LIN {X 0,Y 554.756,Z 744.447,A -85,B 0,C 180,E1 26525.906,E2 26525.906} C_VEL
LIN {X 0,Y 555.497,Z 725.73,A -85,B 0,C 180,E1 26524.354,E2 26524.354} C_VEL
LIN {X 0,Y 556.232,Z 706.632,A -85,B 0,C 180,E1 26523.006,E2 26523.006} C_VEL
LIN {X 0,Y 556.963,Z 686.726,A -85,B 0,C 180,E1 26521.826,E2 26521.826} C_VEL
LIN {X 0,Y 557.64,Z 666.249,A -85,B 0,C 180,E1 26520.833,E2 26520.833} C_VEL
LIN {X 0,Y 558.264,Z 644.541,A -85,B 0,C 180,E1 26519.99,E2 26519.99} C_VEL
LIN {X 0,Y 558.793,Z 623.131,A -85,B 0,C 180,E1 26519.359,E2 26519.359} C_VEL
LIN {X 0,Y 559.115,Z 601.514,A -85,B 0,C 180,E1 26518.923,E2 26518.923} C_VEL
LIN {X 0,Y 560.676,Z 378.924,A -85,B 0,C 180,E1 26515.689,E2 26515.689} C_VEL
LIN {X 0,Y 561.034,Z 312.454,A -85,B 0,C 180,E1 26514.699,E2 26514.699} C_VEL
LIN {X 0,Y 559.13,Z 302.175,A -85,B 0,C 180,E1 26514.381,E2 26514.381} C_VEL
LIN {X 0,Y 560.174,Z 262.496,A -85,B 0,C 180,E1 26511.548,E2 26511.548} C_VEL
LIN {X 0,Y 553.21,Z 246.785,A -85,B 0,C 180,E1 26509.785,E2 26509.785} C_VEL
LIN {X 0,Y 552.322,Z 243.938,A -85,B 0,C 180,E1 26509.493,E2 26509.493} C_VEL
LIN {X 0,Y 552.276,Z 243.94,A -85,B 0,C 180,E1 26506.244,E2 26506.244} C_VEL
LIN {X 0,Y 552.335,Z 243.938,A -85,B 0,C 180,E1 26503.001,E2 26503.001} C_VEL
LIN {X 0,Y 552.275,Z 243.938,A -85,B 0,C 180,E1 26499.858,E2 26499.858} C_VEL
LIN {X 0,Y 552.287,Z 243.939,A -85,B 0,C 180,E1 26496.503,E2 26496.503} C_VEL
LIN {X 0,Y 552.286,Z 243.938,A -85,B 0,C 180,E1 26493.517,E2 26493.517} C_VEL
LIN {X 0,Y 552.27,Z 243.94,A -85,B 0,C 180,E1 26490.22,E2 26490.22} C_VEL
LIN {X 0,Y 552.328,Z 243.939,A -85,B 0,C 180,E1 26487.026,E2 26487.026} C_VEL
LIN {X 0,Y 552.26,Z 243.94,A -85,B 0,C 180,E1 26483.813,E2 26483.813} C_VEL
LIN {X 0,Y 552.351,Z 244.153,A -85,B 0,C 180,E1 26480.713,E2 26480.713} C_VEL
LIN {X 0,Y 553.695,Z 247.553,A -85,B 0,C 180,E1 26480.559,E2 26480.559} C_VEL
LIN {X 0,Y 555.367,Z 250.208,A -85,B 0,C 180,E1 26480.395,E2 26480.395} C_VEL
LIN {X 0,Y 560.988,Z 259.677,A -85,B 0,C 180,E1 26479.842,E2 26479.842} C_VEL
LIN {X 0,Y 559.325,Z 496.337,A -85,B 0,C 180,E1 26476.402,E2 26476.402} C_VEL
LIN {X 0,Y 558.983,Z 531.842,A -85,B 0,C 180,E1 26475.851,E2 26475.851} C_VEL
LIN {X 0,Y 558.554,Z 554.111,A -85,B 0,C 180,E1 26475.298,E2 26475.298} C_VEL
LIN {X 0,Y 557.962,Z 575.135,A -85,B 0,C 180,E1 26474.584,E2 26474.584} C_VEL
LIN {X 0,Y 557.322,Z 596.603,A -85,B 0,C 180,E1 26473.647,E2 26473.647} C_VEL
LIN {X 0,Y 556.604,Z 616.891,A -85,B 0,C 180,E1 26472.555,E2 26472.555} C_VEL
LIN {X 0,Y 555.878,Z 636.118,A -85,B 0,C 180,E1 26471.308,E2 26471.308} C_VEL
LIN {X 0,Y 555.13,Z 655.149,A -85,B 0,C 180,E1 26469.853,E2 26469.853} C_VEL
LIN {X 0,Y 554.42,Z 673.135,A -85,B 0,C 180,E1 26468.244,E2 26468.244} C_VEL
LIN {X 0,Y 553.808,Z 689.545,A -85,B 0,C 180,E1 26466.532,E2 26466.532} C_VEL
LIN {X 0,Y 553.233,Z 705.705,A -85,B 0,C 180,E1 26464.562,E2 26464.562} C_VEL
LIN {X 0,Y 552.797,Z 719.52,A -85,B 0,C 180,E1 26462.593,E2 26462.593} C_VEL
LIN {X 0,Y 552.451,Z 732.51,A -85,B 0,C 180,E1 26460.416,E2 26460.416} C_VEL
LIN {X 0,Y 552.222,Z 742.951,A -85,B 0,C 180,E1 26458.341,E2 26458.341} C_VEL
LIN {X 0,Y 552.065,Z 752.001,A -85,B 0,C 180,E1 26456.159,E2 26456.159} C_VEL
LIN {X 0,Y 551.98,Z 759.324,A -85,B 0,C 180,E1 26453.968,E2 26453.968} C_VEL
LIN {X 0,Y 551.934,Z 765.028,A -85,B 0,C 180,E1 26451.774,E2 26451.774} C_VEL
LIN {X 0,Y 551.912,Z 769.059,A -85,B 0,C 180,E1 26449.564,E2 26449.564} C_VEL
LIN {X 0,Y 551.914,Z 771.636,A -85,B 0,C 180,E1 26447.233,E2 26447.233} C_VEL
LIN {X 0,Y 551.917,Z 772.498,A -85,B 0,C 180,E1 26444.988,E2 26444.988} C_VEL
LIN {X 0,Y 551.911,Z 771.649,A -85,B 0,C 180,E1 26442.695,E2 26442.695} C_VEL
LIN {X 0,Y 551.919,Z 769.139,A -85,B 0,C 180,E1 26440.397,E2 26440.397} C_VEL
LIN {X 0,Y 551.937,Z 765.18,A -85,B 0,C 180,E1 26438.202,E2 26438.202} C_VEL
LIN {X 0,Y 551.98,Z 759.253,A -85,B 0,C 180,E1 26435.917,E2 26435.917} C_VEL
LIN {X 0,Y 552.069,Z 751.656,A -85,B 0,C 180,E1 26433.661,E2 26433.661} C_VEL
LIN {X 0,Y 552.082,Z 750.625,A -85,B 0,C 180,E1 26433.393,E2 26433.393} C_VEL
LIN {X 0,Y 551.135,Z 747.773,A -85,B 0,C 180,E1 26432.65,E2 26432.65} C_VEL
LIN {X 0,Y 545.095,Z 739.69,A -85,B 0,C 180,E1 26430.691,E2 26430.691} C_VEL
LIN {X 0,Y 544.423,Z 736.731,A -85,B 0,C 180,E1 26430.065,E2 26430.065} C_VEL
LIN {X 0,Y 544.761,Z 725.174,A -85,B 0,C 180,E1 26427.968,E2 26427.968} C_VEL
LIN {X 0,Y 545.246,Z 711.568,A -85,B 0,C 180,E1 26425.868,E2 26425.868} C_VEL
LIN {X 0,Y 545.854,Z 696.307,A -85,B 0,C 180,E1 26423.859,E2 26423.859} C_VEL
LIN {X 0,Y 546.544,Z 680.23,A -85,B 0,C 180,E1 26422.044,E2 26422.044} C_VEL
LIN {X 0,Y 547.342,Z 662.41,A -85,B 0,C 180,E1 26420.32,E2 26420.32} C_VEL
LIN {X 0,Y 548.174,Z 644.266,A -85,B 0,C 180,E1 26418.821,E2 26418.821} C_VEL
LIN {X 0,Y 549.064,Z 624.441,A -85,B 0,C 180,E1 26417.432,E2 26417.432} C_VEL
LIN {X 0,Y 549.929,Z 603.469,A -85,B 0,C 180,E1 26416.205,E2 26416.205} C_VEL
LIN {X 0,Y 550.725,Z 582.729,A -85,B 0,C 180,E1 26415.22,E2 26415.22} C_VEL
LIN {X 0,Y 551.396,Z 561.172,A -85,B 0,C 180,E1 26414.411,E2 26414.411} C_VEL
LIN {X 0,Y 551.948,Z 539.46,A -85,B 0,C 180,E1 26413.8,E2 26413.8} C_VEL
LIN {X 0,Y 552.347,Z 516.378,A -85,B 0,C 180,E1 26413.364,E2 26413.364} C_VEL
LIN {X 0,Y 554.178,Z 289.23,A -85,B 0,C 180,E1 26410.034,E2 26410.034} C_VEL
LIN {X 0,Y 554.28,Z 262.154,A -85,B 0,C 180,E1 26409.621,E2 26409.621} C_VEL
LIN {X 0,Y 546.205,Z 249.081,A -85,B 0,C 180,E1 26408.81,E2 26408.81} C_VEL
LIN {X 0,Y 544.543,Z 245.843,A -85,B 0,C 180,E1 26408.631,E2 26408.631} C_VEL
LIN {X 0,Y 544.367,Z 244.904,A -85,B 0,C 180,E1 26408.571,E2 26408.571} C_VEL
LIN {X 0,Y 544.403,Z 244.915,A -85,B 0,C 180,E1 26405.19,E2 26405.19} C_VEL
LIN {X 0,Y 544.372,Z 244.923,A -85,B 0,C 180,E1 26401.937,E2 26401.937} C_VEL
LIN {X 0,Y 544.371,Z 244.926,A -85,B 0,C 180,E1 26398.526,E2 26398.526} C_VEL
LIN {X 0,Y 544.404,Z 244.923,A -85,B 0,C 180,E1 26395.221,E2 26395.221} C_VEL
LIN {X 0,Y 544.364,Z 244.922,A -85,B 0,C 180,E1 26391.893,E2 26391.893} C_VEL
LIN {X 0,Y 544.37,Z 244.925,A -85,B 0,C 180,E1 26388.417,E2 26388.417} C_VEL
LIN {X 0,Y 544.405,Z 244.921,A -85,B 0,C 180,E1 26385.118,E2 26385.118} C_VEL
LIN {X 0,Y 544.358,Z 244.922,A -85,B 0,C 180,E1 26381.872,E2 26381.872} C_VEL
LIN {X 0,Y 544.388,Z 244.924,A -85,B 0,C 180,E1 26378.557,E2 26378.557} C_VEL
LIN {X 0,Y 544.384,Z 244.919,A -85,B 0,C 180,E1 26375.27,E2 26375.27} C_VEL
LIN {X 0,Y 544.352,Z 244.922,A -85,B 0,C 180,E1 26371.896,E2 26371.896} C_VEL
LIN {X 0,Y 544.401,Z 244.922,A -85,B 0,C 180,E1 26368.633,E2 26368.633} C_VEL
LIN {X 0,Y 544.361,Z 244.918,A -85,B 0,C 180,E1 26365.366,E2 26365.366} C_VEL
LIN {X 0,Y 544.356,Z 244.922,A -85,B 0,C 180,E1 26361.977,E2 26361.977} C_VEL
LIN {X 0,Y 544.405,Z 244.922,A -85,B 0,C 180,E1 26358.668,E2 26358.668} C_VEL
LIN {X 0,Y 544.347,Z 244.922,A -85,B 0,C 180,E1 26355.427,E2 26355.427} C_VEL
LIN {X 0,Y 544.366,Z 244.925,A -85,B 0,C 180,E1 26352.028,E2 26352.028} C_VEL
LIN {X 0,Y 544.385,Z 244.921,A -85,B 0,C 180,E1 26348.789,E2 26348.789} C_VEL
LIN {X 0,Y 544.343,Z 244.923,A -85,B 0,C 180,E1 26345.475,E2 26345.475} C_VEL
LIN {X 0,Y 544.393,Z 244.924,A -85,B 0,C 180,E1 26342.194,E2 26342.194} C_VEL
LIN {X 0,Y 544.348,Z 244.924,A -85,B 0,C 180,E1 26339.051,E2 26339.051} C_VEL
LIN {X 0,Y 544.344,Z 244.926,A -85,B 0,C 180,E1 26335.556,E2 26335.556} C_VEL
LIN {X 0,Y 544.402,Z 244.922,A -85,B 0,C 180,E1 26332.297,E2 26332.297} C_VEL
LIN {X 0,Y 544.336,Z 244.924,A -85,B 0,C 180,E1 26329.165,E2 26329.165} C_VEL
LIN {X 0,Y 544.381,Z 244.927,A -85,B 0,C 180,E1 26325.887,E2 26325.887} C_VEL
LIN {X 0,Y 544.35,Z 244.924,A -85,B 0,C 180,E1 26322.667,E2 26322.667} C_VEL
LIN {X 0,Y 544.337,Z 244.924,A -85,B 0,C 180,E1 26319.321,E2 26319.321} C_VEL
LIN {X 0,Y 544.394,Z 244.926,A -85,B 0,C 180,E1 26316.123,E2 26316.123} C_VEL
LIN {X 0,Y 544.329,Z 244.926,A -85,B 0,C 180,E1 26312.921,E2 26312.921} C_VEL
LIN {X 0,Y 544.367,Z 244.926,A -85,B 0,C 180,E1 26309.607,E2 26309.607} C_VEL
LIN {X 0,Y 544.339,Z 244.925,A -85,B 0,C 180,E1 26306.507,E2 26306.507} C_VEL
LIN {X 0,Y 544.333,Z 244.926,A -85,B 0,C 180,E1 26303.145,E2 26303.145} C_VEL
LIN {X 0,Y 544.38,Z 244.925,A -85,B 0,C 180,E1 26299.974,E2 26299.974} C_VEL
LIN {X 0,Y 544.322,Z 244.926,A -85,B 0,C 180,E1 26296.76,E2 26296.76} C_VEL
LIN {X 0,Y 544.386,Z 244.927,A -85,B 0,C 180,E1 26293.595,E2 26293.595} C_VEL
LIN {X 0,Y 544.326,Z 244.925,A -85,B 0,C 180,E1 26290.369,E2 26290.369} C_VEL
LIN {X 0,Y 544.328,Z 244.926,A -85,B 0,C 180,E1 26286.962,E2 26286.962} C_VEL
LIN {X 0,Y 544.368,Z 244.927,A -85,B 0,C 180,E1 26283.79,E2 26283.79} C_VEL
LIN {X 0,Y 544.319,Z 244.925,A -85,B 0,C 180,E1 26280.63,E2 26280.63} C_VEL
LIN {X 0,Y 544.389,Z 244.926,A -85,B 0,C 180,E1 26277.472,E2 26277.472} C_VEL
LIN {X 0,Y 544.325,Z 244.925,A -85,B 0,C 180,E1 26274.2,E2 26274.2} C_VEL
LIN {X 0,Y 544.339,Z 244.926,A -85,B 0,C 180,E1 26270.803,E2 26270.803} C_VEL
LIN {X 0,Y 544.358,Z 244.926,A -85,B 0,C 180,E1 26267.697,E2 26267.697} C_VEL
LIN {X 0,Y 544.327,Z 244.926,A -85,B 0,C 180,E1 26264.443,E2 26264.443} C_VEL
LIN {X 0,Y 544.396,Z 244.924,A -85,B 0,C 180,E1 26261.251,E2 26261.251} C_VEL
LIN {X 0,Y 544.331,Z 244.925,A -85,B 0,C 180,E1 26257.992,E2 26257.992} C_VEL
LIN {X 0,Y 544.351,Z 244.924,A -85,B 0,C 180,E1 26254.645,E2 26254.645} C_VEL
LIN {X 0,Y 544.352,Z 244.926,A -85,B 0,C 180,E1 26251.592,E2 26251.592} C_VEL
LIN {X 0,Y 544.337,Z 244.926,A -85,B 0,C 180,E1 26248.258,E2 26248.258} C_VEL
LIN {X 0,Y 544.405,Z 244.925,A -85,B 0,C 180,E1 26244.995,E2 26244.995} C_VEL
LIN {X 0,Y 544.339,Z 244.926,A -85,B 0,C 180,E1 26241.755,E2 26241.755} C_VEL
LIN {X 0,Y 544.354,Z 244.927,A -85,B 0,C 180,E1 26238.378,E2 26238.378} C_VEL
LIN {X 0,Y 544.381,Z 244.929,A -85,B 0,C 180,E1 26235.147,E2 26235.147} C_VEL
LIN {X 0,Y 544.34,Z 244.929,A -85,B 0,C 180,E1 26231.816,E2 26231.816} C_VEL
LIN {X 0,Y 544.395,Z 245.017,A -85,B 0,C 180,E1 26231.093,E2 26231.093} C_VEL
LIN {X 0,Y 548.823,Z 255.605,A -85,B 0,C 180,E1 26229.915,E2 26229.915} C_VEL
LIN {X 0,Y 553.412,Z 266.114,A -85,B 0,C 180,E1 26228.734,E2 26228.734} C_VEL
LIN {X 0,Y 552.412,Z 303.163,A -85,B 0,C 180,E1 26226.083,E2 26226.083} C_VEL
LIN {X 0,Y 554.642,Z 315.9,A -85,B 0,C 180,E1 26225.716,E2 26225.716} C_VEL
LIN {X 0,Y 552.802,Z 536.145,A -85,B 0,C 180,E1 26222.466,E2 26222.466} C_VEL
LIN {X 0,Y 552.177,Z 609.441,A -85,B 0,C 180,E1 26221.37,E2 26221.37} C_VEL
LIN {X 0,Y 551.642,Z 631.09,A -85,B 0,C 180,E1 26220.851,E2 26220.851} C_VEL
LIN {X 0,Y 551.021,Z 653.26,A -85,B 0,C 180,E1 26220.113,E2 26220.113} C_VEL
LIN {X 0,Y 550.331,Z 673.419,A -85,B 0,C 180,E1 26219.255,E2 26219.255} C_VEL
LIN {X 0,Y 549.499,Z 693.774,A -85,B 0,C 180,E1 26218.174,E2 26218.174} C_VEL
LIN {X 0,Y 548.621,Z 714.159,A -85,B 0,C 180,E1 26216.869,E2 26216.869} C_VEL
LIN {X 0,Y 547.765,Z 732.883,A -85,B 0,C 180,E1 26215.45,E2 26215.45} C_VEL
LIN {X 0,Y 546.978,Z 750.522,A -85,B 0,C 180,E1 26213.883,E2 26213.883} C_VEL
LIN {X 0,Y 546.248,Z 766.698,A -85,B 0,C 180,E1 26212.207,E2 26212.207} C_VEL
LIN {X 0,Y 545.572,Z 782.882,A -85,B 0,C 180,E1 26210.264,E2 26210.264} C_VEL
LIN {X 0,Y 545.042,Z 797.053,A -85,B 0,C 180,E1 26208.281,E2 26208.281} C_VEL
LIN {X 0,Y 544.625,Z 809.74,A -85,B 0,C 180,E1 26206.202,E2 26206.202} C_VEL
LIN {X 0,Y 544.322,Z 820.534,A -85,B 0,C 180,E1 26204.099,E2 26204.099} C_VEL
LIN {X 0,Y 544.119,Z 830.074,A -85,B 0,C 180,E1 26201.876,E2 26201.876} C_VEL
LIN {X 0,Y 544.002,Z 837.94,A -85,B 0,C 180,E1 26199.627,E2 26199.627} C_VEL
LIN {X 0,Y 543.941,Z 843.91,A -85,B 0,C 180,E1 26197.392,E2 26197.392} C_VEL
LIN {X 0,Y 543.921,Z 848.466,A -85,B 0,C 180,E1 26195.061,E2 26195.061} C_VEL
LIN {X 0,Y 543.91,Z 851.236,A -85,B 0,C 180,E1 26192.844,E2 26192.844} C_VEL
LIN {X 0,Y 543.899,Z 852.373,A -85,B 0,C 180,E1 26190.631,E2 26190.631} C_VEL
LIN {X 0,Y 543.899,Z 852.015,A -85,B 0,C 180,E1 26188.313,E2 26188.313} C_VEL
LIN {X 0,Y 543.906,Z 850.219,A -85,B 0,C 180,E1 26186.204,E2 26186.204} C_VEL
LIN {X 0,Y 543.925,Z 846.601,A -85,B 0,C 180,E1 26183.879,E2 26183.879} C_VEL
LIN {X 0,Y 543.965,Z 841.58,A -85,B 0,C 180,E1 26181.65,E2 26181.65} C_VEL
LIN {X 0,Y 544.041,Z 835.043,A -85,B 0,C 180,E1 26179.496,E2 26179.496} C_VEL
LIN {X 0,Y 544.194,Z 826.137,A -85,B 0,C 180,E1 26177.154,E2 26177.154} C_VEL
LIN {X 0,Y 544.438,Z 816.112,A -85,B 0,C 180,E1 26174.992,E2 26174.992} C_VEL
LIN {X 0,Y 544.779,Z 804.625,A -85,B 0,C 180,E1 26172.922,E2 26172.922} C_VEL
LIN {X 0,Y 545.233,Z 791.785,A -85,B 0,C 180,E1 26170.948,E2 26170.948} C_VEL
LIN {X 0,Y 545.792,Z 777.648,A -85,B 0,C 180,E1 26169.069,E2 26169.069} C_VEL
LIN {X 0,Y 546.482,Z 761.672,A -85,B 0,C 180,E1 26167.24,E2 26167.24} C_VEL
LIN {X 0,Y 547.232,Z 744.445,A -85,B 0,C 180,E1 26165.553,E2 26165.553} C_VEL
LIN {X 0,Y 548.104,Z 725.658,A -85,B 0,C 180,E1 26163.977,E2 26163.977} C_VEL
LIN {X 0,Y 548.959,Z 706.635,A -85,B 0,C 180,E1 26162.619,E2 26162.619} C_VEL
LIN {X 0,Y 549.764,Z 687.244,A -85,B 0,C 180,E1 26161.454,E2 26161.454} C_VEL
LIN {X 0,Y 550.55,Z 666.868,A -85,B 0,C 180,E1 26160.449,E2 26160.449} C_VEL
LIN {X 0,Y 551.261,Z 645.621,A -85,B 0,C 180,E1 26159.606,E2 26159.606} C_VEL
LIN {X 0,Y 551.832,Z 624.803,A -85,B 0,C 180,E1 26158.978,E2 26158.978} C_VEL
LIN {X 0,Y 552.243,Z 602.978,A -85,B 0,C 180,E1 26158.519,E2 26158.519} C_VEL
LIN {X 0,Y 554.054,Z 380.884,A -85,B 0,C 180,E1 26155.251,E2 26155.251} C_VEL
LIN {X 0,Y 554.471,Z 313.922,A -85,B 0,C 180,E1 26154.24,E2 26154.24} C_VEL
LIN {X 0,Y 552.308,Z 302.396,A -85,B 0,C 180,E1 26153.888,E2 26153.888} C_VEL
LIN {X 0,Y 553.412,Z 266.114,A -85,B 0,C 180,E1 26151.266,E2 26151.266} C_VEL
LIN {X 0,Y 548.725,Z 255.516,A -85,B 0,C 180,E1 26150.097,E2 26150.097} C_VEL
LIN {X 0,Y 544.489,Z 245.476,A -85,B 0,C 180,E1 26149.092,E2 26149.092} C_VEL
LIN {X 0,Y 544.394,Z 244.927,A -85,B 0,C 180,E1 26149.014,E2 26149.014} C_VEL
LIN {X 0,Y 544.35,Z 244.928,A -85,B 0,C 180,E1 26145.754,E2 26145.754} C_VEL
LIN {X 0,Y 544.34,Z 244.929,A -85,B 0,C 180,E1 26142.386,E2 26142.386} C_VEL
LIN {X 0,Y 544.398,Z 244.926,A -85,B 0,C 180,E1 26139.184,E2 26139.184} C_VEL
LIN {X 0,Y 544.332,Z 244.928,A -85,B 0,C 180,E1 26135.898,E2 26135.898} C_VEL
LIN {X 0,Y 544.352,Z 244.929,A -85,B 0,C 180,E1 26132.532,E2 26132.532} C_VEL
LIN {X 0,Y 544.345,Z 244.929,A -85,B 0,C 180,E1 26129.465,E2 26129.465} C_VEL
LIN {X 0,Y 544.328,Z 244.93,A -85,B 0,C 180,E1 26126.159,E2 26126.159} C_VEL
LIN {X 0,Y 544.395,Z 244.927,A -85,B 0,C 180,E1 26122.916,E2 26122.916} C_VEL
LIN {X 0,Y 544.377,Z 245.171,A -85,B 0,C 180,E1 26121.303,E2 26121.303} C_VEL
LIN {X 0,Y 545.785,Z 248.582,A -85,B 0,C 180,E1 26121.14,E2 26121.14} C_VEL
LIN {X 0,Y 547.429,Z 251.037,A -85,B 0,C 180,E1 26120.975,E2 26120.975} C_VEL
LIN {X 0,Y 554.403,Z 262.797,A -85,B 0,C 180,E1 26120.27,E2 26120.27} C_VEL
LIN {X 0,Y 552.475,Z 500.076,A -85,B 0,C 180,E1 26116.781,E2 26116.781} C_VEL
LIN {X 0,Y 552.096,Z 532.411,A -85,B 0,C 180,E1 26116.266,E2 26116.266} C_VEL
LIN {X 0,Y 551.595,Z 554.888,A -85,B 0,C 180,E1 26115.698,E2 26115.698} C_VEL
LIN {X 0,Y 550.916,Z 576.092,A -85,B 0,C 180,E1 26114.963,E2 26114.963} C_VEL
LIN {X 0,Y 550.195,Z 596.838,A -85,B 0,C 180,E1 26114.042,E2 26114.042} C_VEL
LIN {X 0,Y 549.368,Z 617.108,A -85,B 0,C 180,E1 26112.937,E2 26112.937} C_VEL
LIN {X 0,Y 548.502,Z 637.055,A -85,B 0,C 180,E1 26111.622,E2 26111.622} C_VEL
LIN {X 0,Y 547.634,Z 655.942,A -85,B 0,C 180,E1 26110.149,E2 26110.149} C_VEL
LIN {X 0,Y 546.795,Z 674.342,A -85,B 0,C 180,E1 26108.466,E2 26108.466} C_VEL
LIN {X 0,Y 546.093,Z 690.578,A -85,B 0,C 180,E1 26106.731,E2 26106.731} C_VEL
LIN {X 0,Y 545.437,Z 706.62,A -85,B 0,C 180,E1 26104.733,E2 26104.733} C_VEL
LIN {X 0,Y 544.931,Z 720.295,A -85,B 0,C 180,E1 26102.736,E2 26102.736} C_VEL
LIN {X 0,Y 544.544,Z 732.587,A -85,B 0,C 180,E1 26100.633,E2 26100.633} C_VEL
LIN {X 0,Y 544.266,Z 743.479,A -85,B 0,C 180,E1 26098.422,E2 26098.422} C_VEL
LIN {X 0,Y 544.088,Z 752.449,A -85,B 0,C 180,E1 26096.208,E2 26096.208} C_VEL
LIN {X 0,Y 543.986,Z 759.844,A -85,B 0,C 180,E1 26093.92,E2 26093.92} C_VEL
LIN {X 0,Y 543.939,Z 765.497,A -85,B 0,C 180,E1 26091.652,E2 26091.652} C_VEL
LIN {X 0,Y 543.917,Z 769.397,A -85,B 0,C 180,E1 26089.409,E2 26089.409} C_VEL
LIN {X 0,Y 543.908,Z 771.782,A -85,B 0,C 180,E1 26087.042,E2 26087.042} C_VEL
LIN {X 0,Y 543.905,Z 772.474,A -85,B 0,C 180,E1 26084.761,E2 26084.761} C_VEL
LIN {X 0,Y 543.907,Z 771.513,A -85,B 0,C 180,E1 26082.455,E2 26082.455} C_VEL
LIN {X 0,Y 543.918,Z 768.828,A -85,B 0,C 180,E1 26080.12,E2 26080.12} C_VEL
LIN {X 0,Y 543.933,Z 764.644,A -85,B 0,C 180,E1 26077.865,E2 26077.865} C_VEL
LIN {X 0,Y 543.992,Z 758.658,A -85,B 0,C 180,E1 26075.574,E2 26075.574} C_VEL
LIN {X 0,Y 544.106,Z 751.164,A -85,B 0,C 180,E1 26073.363,E2 26073.363} C_VEL
LIN {X 0,Y 544.301,Z 741.783,A -85,B 0,C 180,E1 26071.113,E2 26071.113} C_VEL
LIN {X 0,Y 544.423,Z 736.731,A -85,B 0,C 180,E1 26070.065,E2 26070.065} C_VEL
LIN {X 0,Y 543.541,Z 733.191,A -85,B 0,C 180,E1 26069.343,E2 26069.343} C_VEL
LIN {X 0,Y 537.721,Z 723.441,A -85,B 0,C 180,E1 26067.437,E2 26067.437} C_VEL
LIN {X 0,Y 537.11,Z 719.871,A -85,B 0,C 180,E1 26066.839,E2 26066.839} C_VEL
LIN {X 0,Y 537.708,Z 706.045,A -85,B 0,C 180,E1 26064.802,E2 26064.802} C_VEL
LIN {X 0,Y 538.457,Z 690.185,A -85,B 0,C 180,E1 26062.808,E2 26062.808} C_VEL
LIN {X 0,Y 539.317,Z 673.099,A -85,B 0,C 180,E1 26060.969,E2 26060.969} C_VEL
LIN {X 0,Y 540.255,Z 654.693,A -85,B 0,C 180,E1 26059.282,E2 26059.282} C_VEL
LIN {X 0,Y 541.252,Z 635.649,A -85,B 0,C 180,E1 26057.798,E2 26057.798} C_VEL
LIN {X 0,Y 542.197,Z 616.697,A -85,B 0,C 180,E1 26056.544,E2 26056.544} C_VEL
LIN {X 0,Y 543.16,Z 595.704,A -85,B 0,C 180,E1 26055.394,E2 26055.394} C_VEL
LIN {X 0,Y 544.026,Z 574.141,A -85,B 0,C 180,E1 26054.447,E2 26054.447} C_VEL
LIN {X 0,Y 544.72,Z 552.664,A -85,B 0,C 180,E1 26053.712,E2 26053.712} C_VEL
LIN {X 0,Y 545.299,Z 530.695,A -85,B 0,C 180,E1 26053.171,E2 26053.171} C_VEL
LIN {X 0,Y 545.781,Z 488.239,A -85,B 0,C 180,E1 26052.511,E2 26052.511} C_VEL
LIN {X 0,Y 547.822,Z 265.586,A -85,B 0,C 180,E1 26049.195,E2 26049.195} C_VEL
LIN {X 0,Y 538.295,Z 250.11,A -85,B 0,C 180,E1 26048.21,E2 26048.21} C_VEL
LIN {X 0,Y 536.619,Z 246.873,A -85,B 0,C 180,E1 26048.023,E2 26048.023} C_VEL
LIN {X 0,Y 536.434,Z 245.877,A -85,B 0,C 180,E1 26047.965,E2 26047.965} C_VEL
LIN {X 0,Y 536.429,Z 245.916,A -85,B 0,C 180,E1 26044.516,E2 26044.516} C_VEL
LIN {X 0,Y 536.466,Z 245.914,A -85,B 0,C 180,E1 26041.193,E2 26041.193} C_VEL
LIN {X 0,Y 536.432,Z 245.912,A -85,B 0,C 180,E1 26037.895,E2 26037.895} C_VEL
LIN {X 0,Y 536.43,Z 245.915,A -85,B 0,C 180,E1 26034.444,E2 26034.444} C_VEL
LIN {X 0,Y 536.467,Z 245.912,A -85,B 0,C 180,E1 26031.083,E2 26031.083} C_VEL
LIN {X 0,Y 536.427,Z 245.911,A -85,B 0,C 180,E1 26027.746,E2 26027.746} C_VEL
LIN {X 0,Y 536.423,Z 245.911,A -85,B 0,C 180,E1 26024.244,E2 26024.244} C_VEL
LIN {X 0,Y 536.465,Z 245.911,A -85,B 0,C 180,E1 26020.96,E2 26020.96} C_VEL
LIN {X 0,Y 536.417,Z 245.911,A -85,B 0,C 180,E1 26017.714,E2 26017.714} C_VEL
LIN {X 0,Y 536.43,Z 245.913,A -85,B 0,C 180,E1 26014.277,E2 26014.277} C_VEL
LIN {X 0,Y 536.463,Z 245.908,A -85,B 0,C 180,E1 26010.962,E2 26010.962} C_VEL
LIN {X 0,Y 536.414,Z 245.911,A -85,B 0,C 180,E1 26007.651,E2 26007.651} C_VEL
LIN {X 0,Y 536.433,Z 245.913,A -85,B 0,C 180,E1 26004.224,E2 26004.224} C_VEL
LIN {X 0,Y 536.446,Z 245.907,A -85,B 0,C 180,E1 26000.994,E2 26000.994} C_VEL
LIN {X 0,Y 536.409,Z 245.911,A -85,B 0,C 180,E1 25997.623,E2 25997.623} C_VEL
LIN {X 0,Y 536.453,Z 245.912,A -85,B 0,C 180,E1 25994.322,E2 25994.322} C_VEL
LIN {X 0,Y 536.423,Z 245.911,A -85,B 0,C 180,E1 25991.077,E2 25991.077} C_VEL
LIN {X 0,Y 536.407,Z 245.913,A -85,B 0,C 180,E1 25987.652,E2 25987.652} C_VEL
LIN {X 0,Y 536.464,Z 245.913,A -85,B 0,C 180,E1 25984.382,E2 25984.382} C_VEL
LIN {X 0,Y 536.408,Z 245.911,A -85,B 0,C 180,E1 25981.135,E2 25981.135} C_VEL
LIN {X 0,Y 536.409,Z 245.912,A -85,B 0,C 180,E1 25977.66,E2 25977.66} C_VEL
LIN {X 0,Y 536.461,Z 245.914,A -85,B 0,C 180,E1 25974.348,E2 25974.348} C_VEL
LIN {X 0,Y 536.4,Z 245.915,A -85,B 0,C 180,E1 25971.086,E2 25971.086} C_VEL
LIN {X 0,Y 536.419,Z 245.916,A -85,B 0,C 180,E1 25967.712,E2 25967.712} C_VEL
LIN {X 0,Y 536.432,Z 245.913,A -85,B 0,C 180,E1 25964.49,E2 25964.49} C_VEL
LIN {X 0,Y 536.395,Z 245.915,A -85,B 0,C 180,E1 25961.145,E2 25961.145} C_VEL
LIN {X 0,Y 536.458,Z 245.915,A -85,B 0,C 180,E1 25957.953,E2 25957.953} C_VEL
LIN {X 0,Y 536.399,Z 245.911,A -85,B 0,C 180,E1 25954.714,E2 25954.714} C_VEL
LIN {X 0,Y 536.395,Z 245.914,A -85,B 0,C 180,E1 25951.209,E2 25951.209} C_VEL
LIN {X 0,Y 536.454,Z 245.914,A -85,B 0,C 180,E1 25948.011,E2 25948.011} C_VEL
LIN {X 0,Y 536.388,Z 245.913,A -85,B 0,C 180,E1 25944.795,E2 25944.795} C_VEL
LIN {X 0,Y 536.43,Z 245.915,A -85,B 0,C 180,E1 25941.54,E2 25941.54} C_VEL
LIN {X 0,Y 536.398,Z 245.915,A -85,B 0,C 180,E1 25938.36,E2 25938.36} C_VEL
LIN {X 0,Y 536.391,Z 245.915,A -85,B 0,C 180,E1 25935.015,E2 25935.015} C_VEL
LIN {X 0,Y 536.44,Z 245.916,A -85,B 0,C 180,E1 25931.829,E2 25931.829} C_VEL
LIN {X 0,Y 536.38,Z 245.916,A -85,B 0,C 180,E1 25928.575,E2 25928.575} C_VEL
LIN {X 0,Y 536.427,Z 245.916,A -85,B 0,C 180,E1 25925.346,E2 25925.346} C_VEL
LIN {X 0,Y 536.393,Z 245.917,A -85,B 0,C 180,E1 25922.135,E2 25922.135} C_VEL
LIN {X 0,Y 536.385,Z 245.916,A -85,B 0,C 180,E1 25918.717,E2 25918.717} C_VEL
LIN {X 0,Y 536.448,Z 245.917,A -85,B 0,C 180,E1 25915.509,E2 25915.509} C_VEL
LIN {X 0,Y 536.385,Z 245.916,A -85,B 0,C 180,E1 25912.286,E2 25912.286} C_VEL
LIN {X 0,Y 536.414,Z 245.914,A -85,B 0,C 180,E1 25908.93,E2 25908.93} C_VEL
LIN {X 0,Y 536.413,Z 245.915,A -85,B 0,C 180,E1 25905.751,E2 25905.751} C_VEL
LIN {X 0,Y 536.391,Z 245.915,A -85,B 0,C 180,E1 25902.423,E2 25902.423} C_VEL
LIN {X 0,Y 536.458,Z 245.912,A -85,B 0,C 180,E1 25899.145,E2 25899.145} C_VEL
LIN {X 0,Y 536.397,Z 245.914,A -85,B 0,C 180,E1 25895.906,E2 25895.906} C_VEL
LIN {X 0,Y 536.403,Z 245.913,A -85,B 0,C 180,E1 25892.465,E2 25892.465} C_VEL
LIN {X 0,Y 536.452,Z 245.916,A -85,B 0,C 180,E1 25889.227,E2 25889.227} C_VEL
LIN {X 0,Y 536.396,Z 245.916,A -85,B 0,C 180,E1 25885.998,E2 25885.998} C_VEL
LIN {X 0,Y 536.441,Z 245.913,A -85,B 0,C 180,E1 25882.716,E2 25882.716} C_VEL
LIN {X 0,Y 536.41,Z 245.917,A -85,B 0,C 180,E1 25879.558,E2 25879.558} C_VEL
LIN {X 0,Y 536.404,Z 245.918,A -85,B 0,C 180,E1 25876.099,E2 25876.099} C_VEL
LIN {X 0,Y 536.463,Z 245.915,A -85,B 0,C 180,E1 25872.864,E2 25872.864} C_VEL
LIN {X 0,Y 536.404,Z 245.933,A -85,B 0,C 180,E1 25871.715,E2 25871.715} C_VEL
LIN {X 0,Y 537.789,Z 249.492,A -85,B 0,C 180,E1 25871.312,E2 25871.312} C_VEL
LIN {X 0,Y 546.668,Z 269.771,A -85,B 0,C 180,E1 25869.02,E2 25869.02} C_VEL
LIN {X 0,Y 545.621,Z 303.108,A -85,B 0,C 180,E1 25866.605,E2 25866.605} C_VEL
LIN {X 0,Y 548.131,Z 317.548,A -85,B 0,C 180,E1 25866.181,E2 25866.181} C_VEL
LIN {X 0,Y 546.036,Z 538.054,A -85,B 0,C 180,E1 25862.889,E2 25862.889} C_VEL
LIN {X 0,Y 545.342,Z 609.441,A -85,B 0,C 180,E1 25861.809,E2 25861.809} C_VEL
LIN {X 0,Y 544.741,Z 631.09,A -85,B 0,C 180,E1 25861.285,E2 25861.285} C_VEL
LIN {X 0,Y 544.046,Z 653.257,A -85,B 0,C 180,E1 25860.539,E2 25860.539} C_VEL
LIN {X 0,Y 543.253,Z 673.418,A -85,B 0,C 180,E1 25859.674,E2 25859.674} C_VEL
LIN {X 0,Y 542.321,Z 693.777,A -85,B 0,C 180,E1 25858.581,E2 25858.581} C_VEL
LIN {X 0,Y 541.316,Z 714.156,A -85,B 0,C 180,E1 25857.262,E2 25857.262} C_VEL
LIN {X 0,Y 540.362,Z 732.791,A -85,B 0,C 180,E1 25855.832,E2 25855.832} C_VEL
LIN {X 0,Y 539.448,Z 750.621,A -85,B 0,C 180,E1 25854.228,E2 25854.228} C_VEL
LIN {X 0,Y 538.586,Z 767.204,A -85,B 0,C 180,E1 25852.483,E2 25852.483} C_VEL
LIN {X 0,Y 537.832,Z 782.883,A -85,B 0,C 180,E1 25850.569,E2 25850.569} C_VEL
LIN {X 0,Y 537.225,Z 797.054,A -85,B 0,C 180,E1 25848.556,E2 25848.556} C_VEL
LIN {X 0,Y 536.747,Z 809.739,A -85,B 0,C 180,E1 25846.447,E2 25846.447} C_VEL
LIN {X 0,Y 536.402,Z 820.339,A -85,B 0,C 180,E1 25844.353,E2 25844.353} C_VEL
LIN {X 0,Y 536.157,Z 830.074,A -85,B 0,C 180,E1 25842.055,E2 25842.055} C_VEL
LIN {X 0,Y 536.018,Z 837.94,A -85,B 0,C 180,E1 25839.772,E2 25839.772} C_VEL
LIN {X 0,Y 535.945,Z 843.91,A -85,B 0,C 180,E1 25837.503,E2 25837.503} C_VEL
LIN {X 0,Y 535.923,Z 848.465,A -85,B 0,C 180,E1 25835.137,E2 25835.137} C_VEL
LIN {X 0,Y 535.911,Z 851.236,A -85,B 0,C 180,E1 25832.886,E2 25832.886} C_VEL
LIN {X 0,Y 535.899,Z 852.373,A -85,B 0,C 180,E1 25830.64,E2 25830.64} C_VEL
LIN {X 0,Y 535.9,Z 852.015,A -85,B 0,C 180,E1 25828.288,E2 25828.288} C_VEL
LIN {X 0,Y 535.908,Z 850.219,A -85,B 0,C 180,E1 25826.148,E2 25826.148} C_VEL
LIN {X 0,Y 535.926,Z 846.601,A -85,B 0,C 180,E1 25823.787,E2 25823.787} C_VEL
LIN {X 0,Y 535.968,Z 841.58,A -85,B 0,C 180,E1 25821.524,E2 25821.524} C_VEL
LIN {X 0,Y 536.059,Z 835.109,A -85,B 0,C 180,E1 25819.358,E2 25819.358} C_VEL
LIN {X 0,Y 536.233,Z 826.595,A -85,B 0,C 180,E1 25817.07,E2 25817.07} C_VEL
LIN {X 0,Y 536.512,Z 816.682,A -85,B 0,C 180,E1 25814.875,E2 25814.875} C_VEL
LIN {X 0,Y 536.895,Z 805.267,A -85,B 0,C 180,E1 25812.775,E2 25812.775} C_VEL
LIN {X 0,Y 537.446,Z 791.784,A -85,B 0,C 180,E1 25810.661,E2 25810.661} C_VEL
LIN {X 0,Y 538.093,Z 777.647,A -85,B 0,C 180,E1 25808.755,E2 25808.755} C_VEL
LIN {X 0,Y 538.888,Z 761.611,A -85,B 0,C 180,E1 25806.894,E2 25806.894} C_VEL
LIN {X 0,Y 539.74,Z 744.456,A -85,B 0,C 180,E1 25805.192,E2 25805.192} C_VEL
LIN {X 0,Y 540.726,Z 725.655,A -85,B 0,C 180,E1 25803.595,E2 25803.595} C_VEL
LIN {X 0,Y 541.712,Z 706.638,A -85,B 0,C 180,E1 25802.221,E2 25802.221} C_VEL
LIN {X 0,Y 542.582,Z 687.945,A -85,B 0,C 180,E1 25801.083,E2 25801.083} C_VEL
LIN {X 0,Y 543.487,Z 667.479,A -85,B 0,C 180,E1 25800.055,E2 25800.055} C_VEL
LIN {X 0,Y 544.284,Z 646.701,A -85,B 0,C 180,E1 25799.213,E2 25799.213} C_VEL
LIN {X 0,Y 544.919,Z 625.849,A -85,B 0,C 180,E1 25798.571,E2 25798.571} C_VEL
LIN {X 0,Y 545.409,Z 603.622,A -85,B 0,C 180,E1 25798.09,E2 25798.09} C_VEL
LIN {X 0,Y 547.46,Z 383.047,A -85,B 0,C 180,E1 25794.804,E2 25794.804} C_VEL
LIN {X 0,Y 547.95,Z 315.388,A -85,B 0,C 180,E1 25793.771,E2 25793.771} C_VEL
LIN {X 0,Y 545.533,Z 302.117,A -85,B 0,C 180,E1 25793.347,E2 25793.347} C_VEL
LIN {X 0,Y 546.668,Z 269.77,A -85,B 0,C 180,E1 25790.98,E2 25790.98} C_VEL
LIN {X 0,Y 538.015,Z 250.328,A -85,B 0,C 180,E1 25788.984,E2 25788.984} C_VEL
LIN {X 0,Y 536.41,Z 245.92,A -85,B 0,C 180,E1 25788.532,E2 25788.532} C_VEL
LIN {X 0,Y 536.459,Z 245.915,A -85,B 0,C 180,E1 25785.245,E2 25785.245} C_VEL
LIN {X 0,Y 536.398,Z 245.917,A -85,B 0,C 180,E1 25781.948,E2 25781.948} C_VEL
LIN {X 0,Y 536.42,Z 245.918,A -85,B 0,C 180,E1 25778.64,E2 25778.64} C_VEL
LIN {X 0,Y 536.42,Z 245.916,A -85,B 0,C 180,E1 25775.429,E2 25775.429} C_VEL
LIN {X 0,Y 536.39,Z 245.918,A -85,B 0,C 180,E1 25772.091,E2 25772.091} C_VEL
LIN {X 0,Y 536.453,Z 245.916,A -85,B 0,C 180,E1 25768.835,E2 25768.835} C_VEL
LIN {X 0,Y 536.394,Z 245.919,A -85,B 0,C 180,E1 25765.551,E2 25765.551} C_VEL
LIN {X 0,Y 536.388,Z 245.922,A -85,B 0,C 180,E1 25762.113,E2 25762.113} C_VEL
LIN {X 0,Y 536.417,Z 246.171,A -85,B 0,C 180,E1 25761.915,E2 25761.915} C_VEL
LIN {X 0,Y 537.732,Z 249.471,A -85,B 0,C 180,E1 25761.755,E2 25761.755} C_VEL
LIN {X 0,Y 539.482,Z 251.972,A -85,B 0,C 180,E1 25761.576,E2 25761.576} C_VEL
LIN {X 0,Y 547.851,Z 265.911,A -85,B 0,C 180,E1 25760.707,E2 25760.707} C_VEL
LIN {X 0,Y 545.648,Z 504.068,A -85,B 0,C 180,E1 25757.167,E2 25757.167} C_VEL
LIN {X 0,Y 545.234,Z 533.131,A -85,B 0,C 180,E1 25756.689,E2 25756.689} C_VEL
LIN {X 0,Y 544.657,Z 556.001,A -85,B 0,C 180,E1 25756.098,E2 25756.098} C_VEL
LIN {X 0,Y 543.864,Z 577.688,A -85,B 0,C 180,E1 25755.325,E2 25755.325} C_VEL
LIN {X 0,Y 543.047,Z 598.11,A -85,B 0,C 180,E1 25754.394,E2 25754.394} C_VEL
LIN {X 0,Y 542.122,Z 618.21,A -85,B 0,C 180,E1 25753.276,E2 25753.276} C_VEL
LIN {X 0,Y 541.107,Z 638.73,A -85,B 0,C 180,E1 25751.891,E2 25751.891} C_VEL
LIN {X 0,Y 540.125,Z 657.352,A -85,B 0,C 180,E1 25750.399,E2 25750.399} C_VEL
LIN {X 0,Y 539.177,Z 675.532,A -85,B 0,C 180,E1 25748.694,E2 25748.694} C_VEL
LIN {X 0,Y 538.335,Z 692.513,A -85,B 0,C 180,E1 25746.828,E2 25746.828} C_VEL
LIN {X 0,Y 537.641,Z 707.503,A -85,B 0,C 180,E1 25744.909,E2 25744.909} C_VEL
LIN {X 0,Y 537.044,Z 721.721,A -85,B 0,C 180,E1 25742.776,E2 25742.776} C_VEL
LIN {X 0,Y 536.611,Z 733.783,A -85,B 0,C 180,E1 25740.642,E2 25740.642} C_VEL
LIN {X 0,Y 536.287,Z 744.905,A -85,B 0,C 180,E1 25738.292,E2 25738.292} C_VEL
LIN {X 0,Y 536.096,Z 753.636,A -85,B 0,C 180,E1 25736.045,E2 25736.045} C_VEL
LIN {X 0,Y 535.987,Z 760.589,A -85,B 0,C 180,E1 25733.79,E2 25733.79} C_VEL
LIN {X 0,Y 535.936,Z 766.138,A -85,B 0,C 180,E1 25731.418,E2 25731.418} C_VEL
LIN {X 0,Y 535.909,Z 769.851,A -85,B 0,C 180,E1 25729.14,E2 25729.14} C_VEL
LIN {X 0,Y 535.899,Z 771.927,A -85,B 0,C 180,E1 25726.845,E2 25726.845} C_VEL
LIN {X 0,Y 535.906,Z 772.416,A -85,B 0,C 180,E1 25724.417,E2 25724.417} C_VEL
LIN {X 0,Y 535.908,Z 771.247,A -85,B 0,C 180,E1 25722.073,E2 25722.073} C_VEL
LIN {X 0,Y 535.91,Z 768.312,A -85,B 0,C 180,E1 25719.697,E2 25719.697} C_VEL
LIN {X 0,Y 535.939,Z 763.817,A -85,B 0,C 180,E1 25717.401,E2 25717.401} C_VEL
LIN {X 0,Y 536.027,Z 757.576,A -85,B 0,C 180,E1 25715.069,E2 25715.069} C_VEL
LIN {X 0,Y 536.177,Z 749.757,A -85,B 0,C 180,E1 25712.812,E2 25712.812} C_VEL
LIN {X 0,Y 536.424,Z 739.992,A -85,B 0,C 180,E1 25710.525,E2 25710.525} C_VEL
LIN {X 0,Y 536.79,Z 728.673,A -85,B 0,C 180,E1 25708.316,E2 25708.316} C_VEL
LIN {X 0,Y 537.11,Z 719.871,A -85,B 0,C 180,E1 25706.839,E2 25706.839} C_VEL
LIN {X 0,Y 536.295,Z 715.69,A -85,B 0,C 180,E1 25706.149,E2 25706.149} C_VEL
LIN {X 0,Y 530.745,Z 704.443,A -85,B 0,C 180,E1 25704.306,E2 25704.306} C_VEL
LIN {X 0,Y 530.261,Z 700.374,A -85,B 0,C 180,E1 25703.734,E2 25703.734} C_VEL
LIN {X 0,Y 531.123,Z 684.545,A -85,B 0,C 180,E1 25701.827,E2 25701.827} C_VEL
LIN {X 0,Y 532.133,Z 667.051,A -85,B 0,C 180,E1 25700.017,E2 25700.017} C_VEL
LIN {X 0,Y 533.263,Z 648.06,A -85,B 0,C 180,E1 25698.345,E2 25698.345} C_VEL
LIN {X 0,Y 534.358,Z 629.03,A -85,B 0,C 180,E1 25696.927,E2 25696.927} C_VEL
LIN {X 0,Y 535.447,Z 608.76,A -85,B 0,C 180,E1 25695.659,E2 25695.659} C_VEL
LIN {X 0,Y 536.503,Z 587.481,A -85,B 0,C 180,E1 25694.574,E2 25694.574} C_VEL
LIN {X 0,Y 537.422,Z 565.024,A -85,B 0,C 180,E1 25693.666,E2 25693.666} C_VEL
LIN {X 0,Y 538.188,Z 542.413,A -85,B 0,C 180,E1 25692.987,E2 25692.987} C_VEL
LIN {X 0,Y 538.687,Z 520.239,A -85,B 0,C 180,E1 25692.533,E2 25692.533} C_VEL
LIN {X 0,Y 541.031,Z 295.74,A -85,B 0,C 180,E1 25689.161,E2 25689.161} C_VEL
LIN {X 0,Y 541.162,Z 268.343,A -85,B 0,C 180,E1 25688.73,E2 25688.73} C_VEL
LIN {X 0,Y 530.454,Z 251.158,A -85,B 0,C 180,E1 25687.591,E2 25687.591} C_VEL
LIN {X 0,Y 528.732,Z 247.94,A -85,B 0,C 180,E1 25687.393,E2 25687.393} C_VEL
LIN {X 0,Y 528.521,Z 246.855,A -85,B 0,C 180,E1 25687.339,E2 25687.339} C_VEL
LIN {X 0,Y 528.49,Z 246.903,A -85,B 0,C 180,E1 25684.043,E2 25684.043} C_VEL
LIN {X 0,Y 528.497,Z 246.905,A -85,B 0,C 180,E1 25680.593,E2 25680.593} C_VEL
LIN {X 0,Y 528.53,Z 246.901,A -85,B 0,C 180,E1 25677.241,E2 25677.241} C_VEL
LIN {X 0,Y 528.489,Z 246.901,A -85,B 0,C 180,E1 25673.884,E2 25673.884} C_VEL
LIN {X 0,Y 528.488,Z 246.903,A -85,B 0,C 180,E1 25670.373,E2 25670.373} C_VEL
LIN {X 0,Y 528.528,Z 246.901,A -85,B 0,C 180,E1 25667.052,E2 25667.052} C_VEL
LIN {X 0,Y 528.487,Z 246.897,A -85,B 0,C 180,E1 25663.68,E2 25663.68} C_VEL
LIN {X 0,Y 528.486,Z 246.903,A -85,B 0,C 180,E1 25660.245,E2 25660.245} C_VEL
LIN {X 0,Y 528.53,Z 246.9,A -85,B 0,C 180,E1 25656.846,E2 25656.846} C_VEL
LIN {X 0,Y 528.487,Z 246.899,A -85,B 0,C 180,E1 25653.472,E2 25653.472} C_VEL
LIN {X 0,Y 528.479,Z 246.899,A -85,B 0,C 180,E1 25650.001,E2 25650.001} C_VEL
LIN {X 0,Y 528.524,Z 246.902,A -85,B 0,C 180,E1 25646.639,E2 25646.639} C_VEL
LIN {X 0,Y 528.487,Z 246.899,A -85,B 0,C 180,E1 25643.265,E2 25643.265} C_VEL
LIN {X 0,Y 528.475,Z 246.901,A -85,B 0,C 180,E1 25639.867,E2 25639.867} C_VEL
LIN {X 0,Y 528.528,Z 246.901,A -85,B 0,C 180,E1 25636.489,E2 25636.489} C_VEL
LIN {X 0,Y 528.481,Z 246.899,A -85,B 0,C 180,E1 25633.175,E2 25633.175} C_VEL
LIN {X 0,Y 528.471,Z 246.901,A -85,B 0,C 180,E1 25629.744,E2 25629.744} C_VEL
LIN {X 0,Y 528.528,Z 246.9,A -85,B 0,C 180,E1 25626.476,E2 25626.476} C_VEL
LIN {X 0,Y 528.471,Z 246.902,A -85,B 0,C 180,E1 25623.118,E2 25623.118} C_VEL
LIN {X 0,Y 528.469,Z 246.904,A -85,B 0,C 180,E1 25619.621,E2 25619.621} C_VEL
LIN {X 0,Y 528.523,Z 246.899,A -85,B 0,C 180,E1 25616.34,E2 25616.34} C_VEL
LIN {X 0,Y 528.465,Z 246.9,A -85,B 0,C 180,E1 25613.013,E2 25613.013} C_VEL
LIN {X 0,Y 528.468,Z 246.903,A -85,B 0,C 180,E1 25609.512,E2 25609.512} C_VEL
LIN {X 0,Y 528.52,Z 246.903,A -85,B 0,C 180,E1 25606.272,E2 25606.272} C_VEL
LIN {X 0,Y 528.457,Z 246.903,A -85,B 0,C 180,E1 25603.077,E2 25603.077} C_VEL
LIN {X 0,Y 528.491,Z 246.902,A -85,B 0,C 180,E1 25599.749,E2 25599.749} C_VEL
LIN {X 0,Y 528.471,Z 246.904,A -85,B 0,C 180,E1 25596.579,E2 25596.579} C_VEL
LIN {X 0,Y 528.454,Z 246.905,A -85,B 0,C 180,E1 25593.145,E2 25593.145} C_VEL
LIN {X 0,Y 528.515,Z 246.901,A -85,B 0,C 180,E1 25589.836,E2 25589.836} C_VEL
LIN {X 0,Y 528.456,Z 246.903,A -85,B 0,C 180,E1 25586.64,E2 25586.64} C_VEL
LIN {X 0,Y 528.456,Z 246.904,A -85,B 0,C 180,E1 25583.147,E2 25583.147} C_VEL
LIN {X 0,Y 528.508,Z 246.903,A -85,B 0,C 180,E1 25579.907,E2 25579.907} C_VEL
LIN {X 0,Y 528.448,Z 246.904,A -85,B 0,C 180,E1 25576.599,E2 25576.599} C_VEL
LIN {X 0,Y 528.467,Z 246.905,A -85,B 0,C 180,E1 25573.232,E2 25573.232} C_VEL
LIN {X 0,Y 528.475,Z 246.902,A -85,B 0,C 180,E1 25570.022,E2 25570.022} C_VEL
LIN {X 0,Y 528.442,Z 246.904,A -85,B 0,C 180,E1 25566.735,E2 25566.735} C_VEL
LIN {X 0,Y 528.503,Z 246.904,A -85,B 0,C 180,E1 25563.469,E2 25563.469} C_VEL
LIN {X 0,Y 528.448,Z 246.903,A -85,B 0,C 180,E1 25560.215,E2 25560.215} C_VEL
LIN {X 0,Y 528.449,Z 246.905,A -85,B 0,C 180,E1 25556.745,E2 25556.745} C_VEL
LIN {X 0,Y 528.513,Z 246.903,A -85,B 0,C 180,E1 25553.481,E2 25553.481} C_VEL
LIN {X 0,Y 528.449,Z 246.905,A -85,B 0,C 180,E1 25550.194,E2 25550.194} C_VEL
LIN {X 0,Y 528.464,Z 246.903,A -85,B 0,C 180,E1 25546.765,E2 25546.765} C_VEL
LIN {X 0,Y 528.484,Z 246.905,A -85,B 0,C 180,E1 25543.625,E2 25543.625} C_VEL
LIN {X 0,Y 528.451,Z 246.904,A -85,B 0,C 180,E1 25540.318,E2 25540.318} C_VEL
LIN {X 0,Y 528.514,Z 246.901,A -85,B 0,C 180,E1 25537.062,E2 25537.062} C_VEL
LIN {X 0,Y 528.46,Z 246.903,A -85,B 0,C 180,E1 25533.842,E2 25533.842} C_VEL
LIN {X 0,Y 528.463,Z 246.903,A -85,B 0,C 180,E1 25530.408,E2 25530.408} C_VEL
LIN {X 0,Y 528.518,Z 246.903,A -85,B 0,C 180,E1 25527.133,E2 25527.133} C_VEL
LIN {X 0,Y 528.459,Z 246.905,A -85,B 0,C 180,E1 25523.82,E2 25523.82} C_VEL
LIN {X 0,Y 528.473,Z 246.905,A -85,B 0,C 180,E1 25520.354,E2 25520.354} C_VEL
LIN {X 0,Y 528.513,Z 246.906,A -85,B 0,C 180,E1 25517.073,E2 25517.073} C_VEL
LIN {X 0,Y 528.464,Z 246.908,A -85,B 0,C 180,E1 25513.718,E2 25513.718} C_VEL
LIN {X 0,Y 528.504,Z 247.053,A -85,B 0,C 180,E1 25512.336,E2 25512.336} C_VEL
LIN {X 0,Y 529.744,Z 250.352,A -85,B 0,C 180,E1 25511.956,E2 25511.956} C_VEL
LIN {X 0,Y 539.827,Z 273.251,A -85,B 0,C 180,E1 25509.303,E2 25509.303} C_VEL
LIN {X 0,Y 538.89,Z 303.208,A -85,B 0,C 180,E1 25507.137,E2 25507.137} C_VEL
LIN {X 0,Y 541.659,Z 319.017,A -85,B 0,C 180,E1 25506.659,E2 25506.659} C_VEL
LIN {X 0,Y 539.304,Z 539.708,A -85,B 0,C 180,E1 25503.327,E2 25503.327} C_VEL
LIN {X 0,Y 538.541,Z 609.44,A -85,B 0,C 180,E1 25502.259,E2 25502.259} C_VEL
LIN {X 0,Y 537.874,Z 631.088,A -85,B 0,C 180,E1 25501.731,E2 25501.731} C_VEL
LIN {X 0,Y 537.102,Z 653.254,A -85,B 0,C 180,E1 25500.978,E2 25500.978} C_VEL
LIN {X 0,Y 536.193,Z 673.699,A -85,B 0,C 180,E1 25500.09,E2 25500.09} C_VEL
LIN {X 0,Y 535.176,Z 693.681,A -85,B 0,C 180,E1 25499.005,E2 25499.005} C_VEL
LIN {X 0,Y 534.037,Z 714.152,A -85,B 0,C 180,E1 25497.665,E2 25497.665} C_VEL
LIN {X 0,Y 532.934,Z 733.456,A -85,B 0,C 180,E1 25496.159,E2 25496.159} C_VEL
LIN {X 0,Y 531.903,Z 751.374,A -85,B 0,C 180,E1 25494.52,E2 25494.52} C_VEL
LIN {X 0,Y 530.913,Z 768.216,A -85,B 0,C 180,E1 25492.709,E2 25492.709} C_VEL
LIN {X 0,Y 530.066,Z 783.728,A -85,B 0,C 180,E1 25490.769,E2 25490.769} C_VEL
LIN {X 0,Y 529.384,Z 797.763,A -85,B 0,C 180,E1 25488.727,E2 25488.727} C_VEL
LIN {X 0,Y 528.852,Z 810.357,A -85,B 0,C 180,E1 25486.586,E2 25486.586} C_VEL
LIN {X 0,Y 528.448,Z 821.301,A -85,B 0,C 180,E1 25484.364,E2 25484.364} C_VEL
LIN {X 0,Y 528.187,Z 830.483,A -85,B 0,C 180,E1 25482.128,E2 25482.128} C_VEL
LIN {X 0,Y 528.036,Z 837.94,A -85,B 0,C 180,E1 25479.921,E2 25479.921} C_VEL
LIN {X 0,Y 527.955,Z 843.91,A -85,B 0,C 180,E1 25477.617,E2 25477.617} C_VEL
LIN {X 0,Y 527.924,Z 848.465,A -85,B 0,C 180,E1 25475.215,E2 25475.215} C_VEL
LIN {X 0,Y 527.912,Z 851.236,A -85,B 0,C 180,E1 25472.93,E2 25472.93} C_VEL
LIN {X 0,Y 527.899,Z 852.373,A -85,B 0,C 180,E1 25470.65,E2 25470.65} C_VEL
LIN {X 0,Y 527.901,Z 852.015,A -85,B 0,C 180,E1 25468.262,E2 25468.262} C_VEL
LIN {X 0,Y 527.91,Z 850.218,A -85,B 0,C 180,E1 25466.089,E2 25466.089} C_VEL
LIN {X 0,Y 527.926,Z 846.601,A -85,B 0,C 180,E1 25463.692,E2 25463.692} C_VEL
LIN {X 0,Y 527.974,Z 841.58,A -85,B 0,C 180,E1 25461.395,E2 25461.395} C_VEL
LIN {X 0,Y 528.082,Z 835.11,A -85,B 0,C 180,E1 25459.195,E2 25459.195} C_VEL
LIN {X 0,Y 528.285,Z 826.594,A -85,B 0,C 180,E1 25456.872,E2 25456.872} C_VEL
LIN {X 0,Y 528.609,Z 816.681,A -85,B 0,C 180,E1 25454.644,E2 25454.644} C_VEL
LIN {X 0,Y 529.045,Z 805.269,A -85,B 0,C 180,E1 25452.512,E2 25452.512} C_VEL
LIN {X 0,Y 529.665,Z 791.783,A -85,B 0,C 180,E1 25450.365,E2 25450.365} C_VEL
LIN {X 0,Y 530.403,Z 777.646,A -85,B 0,C 180,E1 25448.432,E2 25448.432} C_VEL
LIN {X 0,Y 531.29,Z 761.848,A -85,B 0,C 180,E1 25446.572,E2 25446.572} C_VEL
LIN {X 0,Y 532.24,Z 745.049,A -85,B 0,C 180,E1 25444.876,E2 25444.876} C_VEL
LIN {X 0,Y 533.337,Z 726.386,A -85,B 0,C 180,E1 25443.26,E2 25443.26} C_VEL
LIN {X 0,Y 534.446,Z 707.531,A -85,B 0,C 180,E1 25441.871,E2 25441.871} C_VEL
LIN {X 0,Y 535.475,Z 687.723,A -85,B 0,C 180,E1 25440.649,E2 25440.649} C_VEL
LIN {X 0,Y 536.49,Z 667.148,A -85,B 0,C 180,E1 25439.608,E2 25439.608} C_VEL
LIN {X 0,Y 537.368,Z 646.381,A -85,B 0,C 180,E1 25438.761,E2 25438.761} C_VEL
LIN {X 0,Y 538.082,Z 625.653,A -85,B 0,C 180,E1 25438.119,E2 25438.119} C_VEL
LIN {X 0,Y 538.618,Z 603.428,A -85,B 0,C 180,E1 25437.635,E2 25437.635} C_VEL
LIN {X 0,Y 540.907,Z 384.701,A -85,B 0,C 180,E1 25434.34,E2 25434.34} C_VEL
LIN {X 0,Y 541.495,Z 316.993,A -85,B 0,C 180,E1 25433.295,E2 25433.295} C_VEL
LIN {X 0,Y 538.788,Z 302.079,A -85,B 0,C 180,E1 25432.808,E2 25432.808} C_VEL
LIN {X 0,Y 539.518,Z 278.044,A -85,B 0,C 180,E1 25431.078,E2 25431.078} C_VEL
LIN {X 0,Y 539.46,Z 272.631,A -85,B 0,C 180,E1 25430.69,E2 25430.69} C_VEL
LIN {X 0,Y 531.363,Z 254.47,A -85,B 0,C 180,E1 25428.807,E2 25428.807} C_VEL
LIN {X 0,Y 528.464,Z 246.909,A -85,B 0,C 180,E1 25428.005,E2 25428.005} C_VEL
LIN {X 0,Y 528.475,Z 246.908,A -85,B 0,C 180,E1 25424.582,E2 25424.582} C_VEL
LIN {X 0,Y 528.508,Z 246.905,A -85,B 0,C 180,E1 25421.317,E2 25421.317} C_VEL
LIN {X 0,Y 528.453,Z 246.906,A -85,B 0,C 180,E1 25418.084,E2 25418.084} C_VEL
LIN {X 0,Y 528.502,Z 246.906,A -85,B 0,C 180,E1 25414.807,E2 25414.807} C_VEL
LIN {X 0,Y 528.461,Z 246.907,A -85,B 0,C 180,E1 25411.608,E2 25411.608} C_VEL
LIN {X 0,Y 528.451,Z 246.908,A -85,B 0,C 180,E1 25408.151,E2 25408.151} C_VEL
LIN {X 0,Y 528.51,Z 246.904,A -85,B 0,C 180,E1 25404.835,E2 25404.835} C_VEL
LIN {X 0,Y 528.504,Z 247.075,A -85,B 0,C 180,E1 25402.546,E2 25402.546} C_VEL
LIN {X 0,Y 529.823,Z 250.471,A -85,B 0,C 180,E1 25402.375,E2 25402.375} C_VEL
LIN {X 0,Y 531.563,Z 253.015,A -85,B 0,C 180,E1 25402.193,E2 25402.193} C_VEL
LIN {X 0,Y 541.329,Z 268.961,A -85,B 0,C 180,E1 25401.157,E2 25401.157} C_VEL
LIN {X 0,Y 538.854,Z 506.849,A -85,B 0,C 180,E1 25397.58,E2 25397.58} C_VEL
LIN {X 0,Y 538.402,Z 533.851,A -85,B 0,C 180,E1 25397.123,E2 25397.123} C_VEL
LIN {X 0,Y 537.752,Z 556.764,A -85,B 0,C 180,E1 25396.518,E2 25396.518} C_VEL
LIN {X 0,Y 536.862,Z 578.619,A -85,B 0,C 180,E1 25395.724,E2 25395.724} C_VEL
LIN {X 0,Y 535.919,Z 599.382,A -85,B 0,C 180,E1 25394.755,E2 25394.755} C_VEL
LIN {X 0,Y 534.886,Z 619.256,A -85,B 0,C 180,E1 25393.624,E2 25393.624} C_VEL
LIN {X 0,Y 533.762,Z 639.663,A -85,B 0,C 180,E1 25392.222,E2 25392.222} C_VEL
LIN {X 0,Y 532.623,Z 658.746,A -85,B 0,C 180,E1 25390.657,E2 25390.657} C_VEL
LIN {X 0,Y 531.567,Z 676.723,A -85,B 0,C 180,E1 25388.928,E2 25388.928} C_VEL
LIN {X 0,Y 530.627,Z 693.527,A -85,B 0,C 180,E1 25387.036,E2 25387.036} C_VEL
LIN {X 0,Y 529.846,Z 708.363,A -85,B 0,C 180,E1 25385.09,E2 25385.09} C_VEL
LIN {X 0,Y 529.181,Z 722.478,A -85,B 0,C 180,E1 25382.926,E2 25382.926} C_VEL
LIN {X 0,Y 528.694,Z 734.419,A -85,B 0,C 180,E1 25380.76,E2 25380.76} C_VEL
LIN {X 0,Y 528.343,Z 744.962,A -85,B 0,C 180,E1 25378.483,E2 25378.483} C_VEL
LIN {X 0,Y 528.12,Z 753.852,A -85,B 0,C 180,E1 25376.15,E2 25376.15} C_VEL
LIN {X 0,Y 527.995,Z 760.923,A -85,B 0,C 180,E1 25373.805,E2 25373.805} C_VEL
LIN {X 0,Y 527.942,Z 766.158,A -85,B 0,C 180,E1 25371.507,E2 25371.507} C_VEL
LIN {X 0,Y 527.911,Z 769.861,A -85,B 0,C 180,E1 25369.195,E2 25369.195} C_VEL
LIN {X 0,Y 527.9,Z 771.935,A -85,B 0,C 180,E1 25366.865,E2 25366.865} C_VEL
LIN {X 0,Y 527.903,Z 772.439,A -85,B 0,C 180,E1 25364.513,E2 25364.513} C_VEL
LIN {X 0,Y 527.91,Z 771.334,A -85,B 0,C 180,E1 25362.134,E2 25362.134} C_VEL
LIN {X 0,Y 527.911,Z 768.638,A -85,B 0,C 180,E1 25359.838,E2 25359.838} C_VEL
LIN {X 0,Y 527.943,Z 764.068,A -85,B 0,C 180,E1 25357.392,E2 25357.392} C_VEL
LIN {X 0,Y 528.041,Z 757.906,A -85,B 0,C 180,E1 25355.025,E2 25355.025} C_VEL
LIN {X 0,Y 528.207,Z 750.176,A -85,B 0,C 180,E1 25352.739,E2 25352.739} C_VEL
LIN {X 0,Y 528.485,Z 740.499,A -85,B 0,C 180,E1 25350.412,E2 25350.412} C_VEL
LIN {X 0,Y 528.896,Z 729.264,A -85,B 0,C 180,E1 25348.17,E2 25348.17} C_VEL
LIN {X 0,Y 529.467,Z 716.343,A -85,B 0,C 180,E1 25345.999,E2 25345.999} C_VEL
LIN {X 0,Y 530.178,Z 701.705,A -85,B 0,C 180,E1 25343.912,E2 25343.912} C_VEL
LIN {X 0,Y 530.261,Z 700.374,A -85,B 0,C 180,E1 25343.734,E2 25343.734} C_VEL
LIN {X 0,Y 529.599,Z 695.613,A -85,B 0,C 180,E1 25343.075,E2 25343.075} C_VEL
LIN {X 0,Y 524.368,Z 682.897,A -85,B 0,C 180,E1 25341.314,E2 25341.314} C_VEL
LIN {X 0,Y 523.94,Z 678.322,A -85,B 0,C 180,E1 25340.786,E2 25340.786} C_VEL
LIN {X 0,Y 525.121,Z 660.412,A -85,B 0,C 180,E1 25339.012,E2 25339.012} C_VEL
LIN {X 0,Y 526.393,Z 640.968,A -85,B 0,C 180,E1 25337.382,E2 25337.382} C_VEL
LIN {X 0,Y 527.586,Z 621.686,A -85,B 0,C 180,E1 25336.018,E2 25336.018} C_VEL
LIN {X 0,Y 528.8,Z 601.104,A -85,B 0,C 180,E1 25334.807,E2 25334.807} C_VEL
LIN {X 0,Y 529.916,Z 579.325,A -85,B 0,C 180,E1 25333.769,E2 25333.769} C_VEL
LIN {X 0,Y 530.878,Z 557.04,A -85,B 0,C 180,E1 25332.946,E2 25332.946} C_VEL
LIN {X 0,Y 531.605,Z 534.363,A -85,B 0,C 180,E1 25332.338,E2 25332.338} C_VEL
LIN {X 0,Y 532.101,Z 508.425,A -85,B 0,C 180,E1 25331.888,E2 25331.888} C_VEL
LIN {X 0,Y 534.801,Z 274.974,A -85,B 0,C 180,E1 25328.338,E2 25328.338} C_VEL
LIN {X 0,Y 534.694,Z 271.627,A -85,B 0,C 180,E1 25328.275,E2 25328.275} C_VEL
LIN {X 0,Y 522.669,Z 252.324,A -85,B 0,C 180,E1 25326.954,E2 25326.954} C_VEL
LIN {X 0,Y 520.829,Z 249.144,A -85,B 0,C 180,E1 25326.736,E2 25326.736} C_VEL
LIN {X 0,Y 520.555,Z 247.848,A -85,B 0,C 180,E1 25326.681,E2 25326.681} C_VEL
LIN {X 0,Y 520.589,Z 247.891,A -85,B 0,C 180,E1 25323.32,E2 25323.32} C_VEL
LIN {X 0,Y 520.553,Z 247.89,A -85,B 0,C 180,E1 25319.961,E2 25319.961} C_VEL
LIN {X 0,Y 520.554,Z 247.893,A -85,B 0,C 180,E1 25316.464,E2 25316.464} C_VEL
LIN {X 0,Y 520.59,Z 247.889,A -85,B 0,C 180,E1 25313.068,E2 25313.068} C_VEL
LIN {X 0,Y 520.559,Z 247.889,A -85,B 0,C 180,E1 25309.642,E2 25309.642} C_VEL
LIN {X 0,Y 520.543,Z 247.891,A -85,B 0,C 180,E1 25306.173,E2 25306.173} C_VEL
LIN {X 0,Y 520.585,Z 247.891,A -85,B 0,C 180,E1 25302.761,E2 25302.761} C_VEL
LIN {X 0,Y 520.573,Z 247.888,A -85,B 0,C 180,E1 25299.286,E2 25299.286} C_VEL
LIN {X 0,Y 520.539,Z 247.888,A -85,B 0,C 180,E1 25295.955,E2 25295.955} C_VEL
LIN {X 0,Y 520.574,Z 247.888,A -85,B 0,C 180,E1 25292.533,E2 25292.533} C_VEL
LIN {X 0,Y 520.571,Z 247.885,A -85,B 0,C 180,E1 25289.121,E2 25289.121} C_VEL
LIN {X 0,Y 520.534,Z 247.885,A -85,B 0,C 180,E1 25285.705,E2 25285.705} C_VEL
LIN {X 0,Y 520.561,Z 247.888,A -85,B 0,C 180,E1 25282.274,E2 25282.274} C_VEL
LIN {X 0,Y 520.571,Z 247.887,A -85,B 0,C 180,E1 25278.928,E2 25278.928} C_VEL
LIN {X 0,Y 520.53,Z 247.89,A -85,B 0,C 180,E1 25275.541,E2 25275.541} C_VEL
LIN {X 0,Y 520.556,Z 247.892,A -85,B 0,C 180,E1 25272.104,E2 25272.104} C_VEL
LIN {X 0,Y 520.576,Z 247.887,A -85,B 0,C 180,E1 25268.716,E2 25268.716} C_VEL
LIN {X 0,Y 520.527,Z 247.889,A -85,B 0,C 180,E1 25265.367,E2 25265.367} C_VEL
LIN {X 0,Y 520.549,Z 247.891,A -85,B 0,C 180,E1 25261.929,E2 25261.929} C_VEL
LIN {X 0,Y 520.556,Z 247.891,A -85,B 0,C 180,E1 25258.725,E2 25258.725} C_VEL
LIN {X 0,Y 520.523,Z 247.893,A -85,B 0,C 180,E1 25255.351,E2 25255.351} C_VEL
LIN {X 0,Y 520.576,Z 247.892,A -85,B 0,C 180,E1 25252.078,E2 25252.078} C_VEL
LIN {X 0,Y 520.535,Z 247.89,A -85,B 0,C 180,E1 25248.79,E2 25248.79} C_VEL
LIN {X 0,Y 520.522,Z 247.893,A -85,B 0,C 180,E1 25245.331,E2 25245.331} C_VEL
LIN {X 0,Y 520.578,Z 247.895,A -85,B 0,C 180,E1 25241.989,E2 25241.989} C_VEL
LIN {X 0,Y 520.524,Z 247.889,A -85,B 0,C 180,E1 25238.754,E2 25238.754} C_VEL
LIN {X 0,Y 520.52,Z 247.89,A -85,B 0,C 180,E1 25235.279,E2 25235.279} C_VEL
LIN {X 0,Y 520.58,Z 247.893,A -85,B 0,C 180,E1 25232.01,E2 25232.01} C_VEL
LIN {X 0,Y 520.513,Z 247.892,A -85,B 0,C 180,E1 25228.823,E2 25228.823} C_VEL
LIN {X 0,Y 520.541,Z 247.892,A -85,B 0,C 180,E1 25225.478,E2 25225.478} C_VEL
LIN {X 0,Y 520.54,Z 247.892,A -85,B 0,C 180,E1 25222.211,E2 25222.211} C_VEL
LIN {X 0,Y 520.507,Z 247.893,A -85,B 0,C 180,E1 25218.825,E2 25218.825} C_VEL
LIN {X 0,Y 520.554,Z 247.893,A -85,B 0,C 180,E1 25215.483,E2 25215.483} C_VEL
LIN {X 0,Y 520.523,Z 247.894,A -85,B 0,C 180,E1 25212.197,E2 25212.197} C_VEL
LIN {X 0,Y 520.507,Z 247.895,A -85,B 0,C 180,E1 25208.838,E2 25208.838} C_VEL
LIN {X 0,Y 520.57,Z 247.894,A -85,B 0,C 180,E1 25205.62,E2 25205.62} C_VEL
LIN {X 0,Y 520.506,Z 247.895,A -85,B 0,C 180,E1 25202.31,E2 25202.31} C_VEL
LIN {X 0,Y 520.511,Z 247.894,A -85,B 0,C 180,E1 25198.788,E2 25198.788} C_VEL
LIN {X 0,Y 520.57,Z 247.893,A -85,B 0,C 180,E1 25195.423,E2 25195.423} C_VEL
LIN {X 0,Y 520.512,Z 247.894,A -85,B 0,C 180,E1 25192.16,E2 25192.16} C_VEL
LIN {X 0,Y 520.513,Z 247.892,A -85,B 0,C 180,E1 25188.587,E2 25188.587} C_VEL
LIN {X 0,Y 520.585,Z 247.891,A -85,B 0,C 180,E1 25185.313,E2 25185.313} C_VEL
LIN {X 0,Y 520.518,Z 247.894,A -85,B 0,C 180,E1 25181.954,E2 25181.954} C_VEL
LIN {X 0,Y 520.518,Z 247.892,A -85,B 0,C 180,E1 25178.475,E2 25178.475} C_VEL
LIN {X 0,Y 520.577,Z 247.892,A -85,B 0,C 180,E1 25175.246,E2 25175.246} C_VEL
LIN {X 0,Y 520.517,Z 247.892,A -85,B 0,C 180,E1 25171.925,E2 25171.925} C_VEL
LIN {X 0,Y 520.534,Z 247.893,A -85,B 0,C 180,E1 25168.501,E2 25168.501} C_VEL
LIN {X 0,Y 520.568,Z 247.893,A -85,B 0,C 180,E1 25165.218,E2 25165.218} C_VEL
LIN {X 0,Y 520.52,Z 247.893,A -85,B 0,C 180,E1 25161.931,E2 25161.931} C_VEL
LIN {X 0,Y 520.564,Z 247.894,A -85,B 0,C 180,E1 25158.644,E2 25158.644} C_VEL
LIN {X 0,Y 520.551,Z 247.897,A -85,B 0,C 180,E1 25155.288,E2 25155.288} C_VEL
LIN {X 0,Y 520.579,Z 247.926,A -85,B 0,C 180,E1 25153.005,E2 25153.005} C_VEL
LIN {X 0,Y 521.77,Z 251.209,A -85,B 0,C 180,E1 25152.62,E2 25152.62} C_VEL
LIN {X 0,Y 532.239,Z 274.936,A -85,B 0,C 180,E1 25149.794,E2 25149.794} C_VEL
LIN {X 0,Y 532.958,Z 277.309,A -85,B 0,C 180,E1 25149.55,E2 25149.55} C_VEL
LIN {X 0,Y 532.127,Z 303.085,A -85,B 0,C 180,E1 25147.683,E2 25147.683} C_VEL
LIN {X 0,Y 535.225,Z 320.481,A -85,B 0,C 180,E1 25147.15,E2 25147.15} C_VEL
LIN {X 0,Y 532.614,Z 540.471,A -85,B 0,C 180,E1 25143.79,E2 25143.79} C_VEL
LIN {X 0,Y 531.768,Z 609.627,A -85,B 0,C 180,E1 25142.717,E2 25142.717} C_VEL
LIN {X 0,Y 531.043,Z 631.216,A -85,B 0,C 180,E1 25142.184,E2 25142.184} C_VEL
LIN {X 0,Y 530.189,Z 653.251,A -85,B 0,C 180,E1 25141.427,E2 25141.427} C_VEL
LIN {X 0,Y 529.208,Z 673.414,A -85,B 0,C 180,E1 25140.545,E2 25140.545} C_VEL
LIN {X 0,Y 528.046,Z 693.875,A -85,B 0,C 180,E1 25139.423,E2 25139.423} C_VEL
LIN {X 0,Y 526.793,Z 714.149,A -85,B 0,C 180,E1 25138.079,E2 25138.079} C_VEL
LIN {X 0,Y 525.569,Z 733.453,A -85,B 0,C 180,E1 25136.554,E2 25136.554} C_VEL
LIN {X 0,Y 524.426,Z 751.13,A -85,B 0,C 180,E1 25134.919,E2 25134.919} C_VEL
LIN {X 0,Y 523.334,Z 767.71,A -85,B 0,C 180,E1 25133.116,E2 25133.116} C_VEL
LIN {X 0,Y 522.408,Z 782.882,A -85,B 0,C 180,E1 25131.205,E2 25131.205} C_VEL
LIN {X 0,Y 521.626,Z 797.057,A -85,B 0,C 180,E1 25129.132,E2 25129.132} C_VEL
LIN {X 0,Y 521.011,Z 809.736,A -85,B 0,C 180,E1 25126.958,E2 25126.958} C_VEL
LIN {X 0,Y 520.563,Z 820.337,A -85,B 0,C 180,E1 25124.799,E2 25124.799} C_VEL
LIN {X 0,Y 520.243,Z 830.076,A -85,B 0,C 180,E1 25122.429,E2 25122.429} C_VEL
LIN {X 0,Y 520.066,Z 837.711,A -85,B 0,C 180,E1 25120.149,E2 25120.149} C_VEL
LIN {X 0,Y 519.968,Z 843.656,A -85,B 0,C 180,E1 25117.846,E2 25117.846} C_VEL
LIN {X 0,Y 519.927,Z 848.305,A -85,B 0,C 180,E1 25115.406,E2 25115.406} C_VEL
LIN {X 0,Y 519.916,Z 851.012,A -85,B 0,C 180,E1 25113.196,E2 25113.196} C_VEL
LIN {X 0,Y 519.903,Z 852.351,A -85,B 0,C 180,E1 25110.77,E2 25110.77} C_VEL
LIN {X 0,Y 519.898,Z 852.149,A -85,B 0,C 180,E1 25108.456,E2 25108.456} C_VEL
LIN {X 0,Y 519.909,Z 850.331,A -85,B 0,C 180,E1 25106.139,E2 25106.139} C_VEL
LIN {X 0,Y 519.928,Z 846.807,A -85,B 0,C 180,E1 25103.706,E2 25103.706} C_VEL
LIN {X 0,Y 519.981,Z 841.87,A -85,B 0,C 180,E1 25101.373,E2 25101.373} C_VEL
LIN {X 0,Y 520.1,Z 835.465,A -85,B 0,C 180,E1 25099.14,E2 25099.14} C_VEL
LIN {X 0,Y 520.328,Z 827.052,A -85,B 0,C 180,E1 25096.78,E2 25096.78} C_VEL
LIN {X 0,Y 520.687,Z 817.216,A -85,B 0,C 180,E1 25094.518,E2 25094.518} C_VEL
LIN {X 0,Y 521.174,Z 805.912,A -85,B 0,C 180,E1 25092.354,E2 25092.354} C_VEL
LIN {X 0,Y 521.861,Z 792.547,A -85,B 0,C 180,E1 25090.175,E2 25090.175} C_VEL
LIN {X 0,Y 522.683,Z 778.57,A -85,B 0,C 180,E1 25088.215,E2 25088.215} C_VEL
LIN {X 0,Y 523.677,Z 762.53,A -85,B 0,C 180,E1 25086.291,E2 25086.291} C_VEL
LIN {X 0,Y 524.739,Z 745.931,A -85,B 0,C 180,E1 25084.58,E2 25084.58} C_VEL
LIN {X 0,Y 525.967,Z 727.118,A -85,B 0,C 180,E1 25082.916,E2 25082.916} C_VEL
LIN {X 0,Y 527.2,Z 708.421,A -85,B 0,C 180,E1 25081.511,E2 25081.511} C_VEL
LIN {X 0,Y 528.329,Z 688.724,A -85,B 0,C 180,E1 25080.275,E2 25080.275} C_VEL
LIN {X 0,Y 529.457,Z 668.302,A -85,B 0,C 180,E1 25079.217,E2 25079.217} C_VEL
LIN {X 0,Y 530.441,Z 647.676,A -85,B 0,C 180,E1 25078.353,E2 25078.353} C_VEL
LIN {X 0,Y 531.233,Z 626.589,A -85,B 0,C 180,E1 25077.687,E2 25077.687} C_VEL
LIN {X 0,Y 531.85,Z 604.024,A -85,B 0,C 180,E1 25077.183,E2 25077.183} C_VEL
LIN {X 0,Y 534.39,Z 386.483,A -85,B 0,C 180,E1 25073.866,E2 25073.866} C_VEL
LIN {X 0,Y 535.08,Z 318.651,A -85,B 0,C 180,E1 25072.808,E2 25072.808} C_VEL
LIN {X 0,Y 531.932,Z 301.751,A -85,B 0,C 180,E1 25072.27,E2 25072.27} C_VEL
LIN {X 0,Y 532.46,Z 276.037,A -85,B 0,C 180,E1 25070.462,E2 25070.462} C_VEL
LIN {X 0,Y 524.646,Z 258.374,A -85,B 0,C 180,E1 25068.6,E2 25068.6} C_VEL
LIN {X 0,Y 520.568,Z 247.933,A -85,B 0,C 180,E1 25067.46,E2 25067.46} C_VEL
LIN {X 0,Y 520.52,Z 247.897,A -85,B 0,C 180,E1 25064.076,E2 25064.076} C_VEL
LIN {X 0,Y 520.554,Z 247.896,A -85,B 0,C 180,E1 25060.773,E2 25060.773} C_VEL
LIN {X 0,Y 520.528,Z 247.895,A -85,B 0,C 180,E1 25057.65,E2 25057.65} C_VEL
LIN {X 0,Y 520.517,Z 247.897,A -85,B 0,C 180,E1 25054.252,E2 25054.252} C_VEL
LIN {X 0,Y 520.58,Z 247.893,A -85,B 0,C 180,E1 25050.981,E2 25050.981} C_VEL
LIN {X 0,Y 520.514,Z 247.897,A -85,B 0,C 180,E1 25047.681,E2 25047.681} C_VEL
LIN {X 0,Y 520.512,Z 247.897,A -85,B 0,C 180,E1 25044.153,E2 25044.153} C_VEL
LIN {X 0,Y 520.551,Z 247.982,A -85,B 0,C 180,E1 25043.212,E2 25043.212} C_VEL
LIN {X 0,Y 521.812,Z 251.298,A -85,B 0,C 180,E1 25043.041,E2 25043.041} C_VEL
LIN {X 0,Y 523.703,Z 254.021,A -85,B 0,C 180,E1 25042.828,E2 25042.828} C_VEL
LIN {X 0,Y 534.834,Z 271.974,A -85,B 0,C 180,E1 25041.618,E2 25041.618} C_VEL
LIN {X 0,Y 532.108,Z 507.885,A -85,B 0,C 180,E1 25038.03,E2 25038.03} C_VEL
LIN {X 0,Y 531.618,Z 534.118,A -85,B 0,C 180,E1 25037.578,E2 25037.578} C_VEL
LIN {X 0,Y 530.891,Z 556.992,A -85,B 0,C 180,E1 25036.966,E2 25036.966} C_VEL
LIN {X 0,Y 529.926,Z 578.751,A -85,B 0,C 180,E1 25036.166,E2 25036.166} C_VEL
LIN {X 0,Y 528.869,Z 599.617,A -85,B 0,C 180,E1 25035.181,E2 25035.181} C_VEL
LIN {X 0,Y 527.726,Z 619.457,A -85,B 0,C 180,E1 25034.036,E2 25034.036} C_VEL
LIN {X 0,Y 526.475,Z 639.851,A -85,B 0,C 180,E1 25032.616,E2 25032.616} C_VEL
LIN {X 0,Y 525.166,Z 659.527,A -85,B 0,C 180,E1 25030.977,E2 25030.977} C_VEL
LIN {X 0,Y 524.037,Z 676.874,A -85,B 0,C 180,E1 25029.279,E2 25029.279} C_VEL
LIN {X 0,Y 522.982,Z 693.657,A -85,B 0,C 180,E1 25027.361,E2 25027.361} C_VEL
LIN {X 0,Y 522.101,Z 708.469,A -85,B 0,C 180,E1 25025.386,E2 25025.386} C_VEL
LIN {X 0,Y 521.349,Z 722.57,A -85,B 0,C 180,E1 25023.19,E2 25023.19} C_VEL
LIN {X 0,Y 520.797,Z 734.492,A -85,B 0,C 180,E1 25020.992,E2 25020.992} C_VEL
LIN {X 0,Y 520.402,Z 745.02,A -85,B 0,C 180,E1 25018.68,E2 25018.68} C_VEL
LIN {X 0,Y 520.154,Z 753.714,A -85,B 0,C 180,E1 25016.365,E2 25016.365} C_VEL
LIN {X 0,Y 520.015,Z 760.652,A -85,B 0,C 180,E1 25014.042,E2 25014.042} C_VEL
LIN {X 0,Y 519.946,Z 765.971,A -85,B 0,C 180,E1 25011.709,E2 25011.709} C_VEL
LIN {X 0,Y 519.916,Z 769.767,A -85,B 0,C 180,E1 25009.333,E2 25009.333} C_VEL
LIN {X 0,Y 519.906,Z 771.874,A -85,B 0,C 180,E1 25006.998,E2 25006.998} C_VEL
LIN {X 0,Y 519.902,Z 772.454,A -85,B 0,C 180,E1 25004.611,E2 25004.611} C_VEL
LIN {X 0,Y 519.91,Z 771.409,A -85,B 0,C 180,E1 25002.197,E2 25002.197} C_VEL
LIN {X 0,Y 519.912,Z 768.699,A -85,B 0,C 180,E1 24999.8,E2 24999.8} C_VEL
LIN {X 0,Y 519.955,Z 764.046,A -85,B 0,C 180,E1 24997.264,E2 24997.264} C_VEL
LIN {X 0,Y 520.065,Z 757.867,A -85,B 0,C 180,E1 24994.859,E2 24994.859} C_VEL
LIN {X 0,Y 520.25,Z 750.125,A -85,B 0,C 180,E1 24992.535,E2 24992.535} C_VEL
LIN {X 0,Y 520.564,Z 740.429,A -85,B 0,C 180,E1 24990.17,E2 24990.17} C_VEL
LIN {X 0,Y 521.033,Z 729.17,A -85,B 0,C 180,E1 24987.892,E2 24987.892} C_VEL
LIN {X 0,Y 521.682,Z 716.29,A -85,B 0,C 180,E1 24985.697,E2 24985.697} C_VEL
LIN {X 0,Y 522.493,Z 701.64,A -85,B 0,C 180,E1 24983.578,E2 24983.578} C_VEL
LIN {X 0,Y 523.456,Z 685.927,A -85,B 0,C 180,E1 24981.629,E2 24981.629} C_VEL
LIN {X 0,Y 523.94,Z 678.322,A -85,B 0,C 180,E1 24980.786,E2 24980.786} C_VEL
LIN {X 0,Y 523.365,Z 672.96,A -85,B 0,C 180,E1 24980.176,E2 24980.176} C_VEL
LIN {X 0,Y 518.691,Z 659.701,A -85,B 0,C 180,E1 24978.598,E2 24978.598} C_VEL
LIN {X 0,Y 518.215,Z 653.864,A -85,B 0,C 180,E1 24978.026,E2 24978.026} C_VEL
LIN {X 0,Y 519.534,Z 635.061,A -85,B 0,C 180,E1 24976.515,E2 24976.515} C_VEL
LIN {X 0,Y 520.856,Z 615.892,A -85,B 0,C 180,E1 24975.214,E2 24975.214} C_VEL
LIN {X 0,Y 522.145,Z 594.995,A -85,B 0,C 180,E1 24974.037,E2 24974.037} C_VEL
LIN {X 0,Y 523.34,Z 573.014,A -85,B 0,C 180,E1 24973.052,E2 24973.052} C_VEL
LIN {X 0,Y 524.312,Z 550.379,A -85,B 0,C 180,E1 24972.275,E2 24972.275} C_VEL
LIN {X 0,Y 525.043,Z 528.52,A -85,B 0,C 180,E1 24971.744,E2 24971.744} C_VEL
LIN {X 0,Y 526.652,Z 406.04,A -85,B 0,C 180,E1 24969.846,E2 24969.846} C_VEL
LIN {X 0,Y 528.261,Z 274.718,A -85,B 0,C 180,E1 24967.808,E2 24967.808} C_VEL
LIN {X 0,Y 517.162,Z 257.203,A -85,B 0,C 180,E1 24966.564,E2 24966.564} C_VEL
LIN {X 0,Y 514.842,Z 253.466,A -85,B 0,C 180,E1 24966.289,E2 24966.289} C_VEL
LIN {X 0,Y 512.963,Z 250.398,A -85,B 0,C 180,E1 24966.062,E2 24966.062} C_VEL
LIN {X 0,Y 512.616,Z 248.848,A -85,B 0,C 180,E1 24965.983,E2 24965.983} C_VEL
LIN {X 0,Y 512.613,Z 248.883,A -85,B 0,C 180,E1 24962.439,E2 24962.439} C_VEL
LIN {X 0,Y 512.649,Z 248.881,A -85,B 0,C 180,E1 24959.055,E2 24959.055} C_VEL
LIN {X 0,Y 512.627,Z 248.878,A -85,B 0,C 180,E1 24955.659,E2 24955.659} C_VEL
LIN {X 0,Y 512.606,Z 248.881,A -85,B 0,C 180,E1 24952.236,E2 24952.236} C_VEL
LIN {X 0,Y 512.645,Z 248.879,A -85,B 0,C 180,E1 24948.892,E2 24948.892} C_VEL
LIN {X 0,Y 512.635,Z 248.876,A -85,B 0,C 180,E1 24945.383,E2 24945.383} C_VEL
LIN {X 0,Y 512.603,Z 248.879,A -85,B 0,C 180,E1 24941.933,E2 24941.933} C_VEL
LIN {X 0,Y 512.628,Z 248.879,A -85,B 0,C 180,E1 24938.526,E2 24938.526} C_VEL
LIN {X 0,Y 512.638,Z 248.874,A -85,B 0,C 180,E1 24935.148,E2 24935.148} C_VEL
LIN {X 0,Y 512.598,Z 248.877,A -85,B 0,C 180,E1 24931.79,E2 24931.79} C_VEL
LIN {X 0,Y 512.631,Z 248.879,A -85,B 0,C 180,E1 24928.436,E2 24928.436} C_VEL
LIN {X 0,Y 512.637,Z 248.871,A -85,B 0,C 180,E1 24924.966,E2 24924.966} C_VEL
LIN {X 0,Y 512.595,Z 248.876,A -85,B 0,C 180,E1 24921.589,E2 24921.589} C_VEL
LIN {X 0,Y 512.618,Z 248.879,A -85,B 0,C 180,E1 24918.183,E2 24918.183} C_VEL
LIN {X 0,Y 512.633,Z 248.876,A -85,B 0,C 180,E1 24914.851,E2 24914.851} C_VEL
LIN {X 0,Y 512.592,Z 248.879,A -85,B 0,C 180,E1 24911.431,E2 24911.431} C_VEL
LIN {X 0,Y 512.611,Z 248.881,A -85,B 0,C 180,E1 24908.008,E2 24908.008} C_VEL
LIN {X 0,Y 512.628,Z 248.876,A -85,B 0,C 180,E1 24904.715,E2 24904.715} C_VEL
LIN {X 0,Y 512.588,Z 248.878,A -85,B 0,C 180,E1 24901.326,E2 24901.326} C_VEL
LIN {X 0,Y 512.617,Z 248.878,A -85,B 0,C 180,E1 24897.96,E2 24897.96} C_VEL
LIN {X 0,Y 512.622,Z 248.881,A -85,B 0,C 180,E1 24894.601,E2 24894.601} C_VEL
LIN {X 0,Y 512.583,Z 248.882,A -85,B 0,C 180,E1 24891.235,E2 24891.235} C_VEL
LIN {X 0,Y 512.614,Z 248.883,A -85,B 0,C 180,E1 24887.829,E2 24887.829} C_VEL
LIN {X 0,Y 512.604,Z 248.881,A -85,B 0,C 180,E1 24884.6,E2 24884.6} C_VEL
LIN {X 0,Y 512.579,Z 248.883,A -85,B 0,C 180,E1 24881.156,E2 24881.156} C_VEL
LIN {X 0,Y 512.618,Z 248.884,A -85,B 0,C 180,E1 24877.764,E2 24877.764} C_VEL
LIN {X 0,Y 512.604,Z 248.877,A -85,B 0,C 180,E1 24874.406,E2 24874.406} C_VEL
LIN {X 0,Y 512.575,Z 248.88,A -85,B 0,C 180,E1 24870.993,E2 24870.993} C_VEL
LIN {X 0,Y 512.617,Z 248.882,A -85,B 0,C 180,E1 24867.657,E2 24867.657} C_VEL
LIN {X 0,Y 512.596,Z 248.879,A -85,B 0,C 180,E1 24864.301,E2 24864.301} C_VEL
LIN {X 0,Y 512.571,Z 248.881,A -85,B 0,C 180,E1 24860.912,E2 24860.912} C_VEL
LIN {X 0,Y 512.622,Z 248.881,A -85,B 0,C 180,E1 24857.595,E2 24857.595} C_VEL
LIN {X 0,Y 512.578,Z 248.881,A -85,B 0,C 180,E1 24854.341,E2 24854.341} C_VEL
LIN {X 0,Y 512.57,Z 248.88,A -85,B 0,C 180,E1 24850.905,E2 24850.905} C_VEL
LIN {X 0,Y 512.63,Z 248.88,A -85,B 0,C 180,E1 24847.507,E2 24847.507} C_VEL
LIN {X 0,Y 512.578,Z 248.883,A -85,B 0,C 180,E1 24844.137,E2 24844.137} C_VEL
LIN {X 0,Y 512.566,Z 248.88,A -85,B 0,C 180,E1 24840.669,E2 24840.669} C_VEL
LIN {X 0,Y 512.628,Z 248.881,A -85,B 0,C 180,E1 24837.427,E2 24837.427} C_VEL
LIN {X 0,Y 512.577,Z 248.88,A -85,B 0,C 180,E1 24834.065,E2 24834.065} C_VEL
LIN {X 0,Y 512.572,Z 248.883,A -85,B 0,C 180,E1 24830.568,E2 24830.568} C_VEL
LIN {X 0,Y 512.631,Z 248.88,A -85,B 0,C 180,E1 24827.211,E2 24827.211} C_VEL
LIN {X 0,Y 512.576,Z 248.882,A -85,B 0,C 180,E1 24824.034,E2 24824.034} C_VEL
LIN {X 0,Y 512.58,Z 248.881,A -85,B 0,C 180,E1 24820.514,E2 24820.514} C_VEL
LIN {X 0,Y 512.643,Z 248.878,A -85,B 0,C 180,E1 24817.161,E2 24817.161} C_VEL
LIN {X 0,Y 512.584,Z 248.881,A -85,B 0,C 180,E1 24813.799,E2 24813.799} C_VEL
LIN {X 0,Y 512.582,Z 248.881,A -85,B 0,C 180,E1 24810.299,E2 24810.299} C_VEL
LIN {X 0,Y 512.641,Z 248.88,A -85,B 0,C 180,E1 24806.997,E2 24806.997} C_VEL
LIN {X 0,Y 512.592,Z 248.884,A -85,B 0,C 180,E1 24803.63,E2 24803.63} C_VEL
LIN {X 0,Y 512.589,Z 248.883,A -85,B 0,C 180,E1 24800.22,E2 24800.22} C_VEL
LIN {X 0,Y 512.641,Z 248.883,A -85,B 0,C 180,E1 24796.949,E2 24796.949} C_VEL
LIN {X 0,Y 512.607,Z 249.028,A -85,B 0,C 180,E1 24793.687,E2 24793.687} C_VEL
LIN {X 0,Y 513.81,Z 252.211,A -85,B 0,C 180,E1 24793.298,E2 24793.298} C_VEL
LIN {X 0,Y 522.469,Z 271.789,A -85,B 0,C 180,E1 24790.879,E2 24790.879} C_VEL
LIN {X 0,Y 526.151,Z 280.209,A -85,B 0,C 180,E1 24789.891,E2 24789.891} C_VEL
LIN {X 0,Y 525.313,Z 302.438,A -85,B 0,C 180,E1 24788.255,E2 24788.255} C_VEL
LIN {X 0,Y 528.756,Z 322.024,A -85,B 0,C 180,E1 24787.639,E2 24787.639} C_VEL
LIN {X 0,Y 525.992,Z 538.69,A -85,B 0,C 180,E1 24784.302,E2 24784.302} C_VEL
LIN {X 0,Y 525.036,Z 609.627,A -85,B 0,C 180,E1 24783.19,E2 24783.19} C_VEL
LIN {X 0,Y 524.259,Z 631.084,A -85,B 0,C 180,E1 24782.656,E2 24782.656} C_VEL
LIN {X 0,Y 523.31,Z 653.247,A -85,B 0,C 180,E1 24781.888,E2 24781.888} C_VEL
LIN {X 0,Y 522.24,Z 673.412,A -85,B 0,C 180,E1 24780.997,E2 24780.997} C_VEL
LIN {X 0,Y 520.955,Z 693.881,A -85,B 0,C 180,E1 24779.863,E2 24779.863} C_VEL
LIN {X 0,Y 519.586,Z 714.145,A -85,B 0,C 180,E1 24778.503,E2 24778.503} C_VEL
LIN {X 0,Y 518.23,Z 733.45,A -85,B 0,C 180,E1 24776.961,E2 24776.961} C_VEL
LIN {X 0,Y 516.954,Z 751.13,A -85,B 0,C 180,E1 24775.304,E2 24775.304} C_VEL
LIN {X 0,Y 515.782,Z 767.337,A -85,B 0,C 180,E1 24773.519,E2 24773.519} C_VEL
LIN {X 0,Y 514.699,Z 783.258,A -85,B 0,C 180,E1 24771.485,E2 24771.485} C_VEL
LIN {X 0,Y 513.847,Z 797.059,A -85,B 0,C 180,E1 24769.434,E2 24769.434} C_VEL
LIN {X 0,Y 513.152,Z 809.734,A -85,B 0,C 180,E1 24767.226,E2 24767.226} C_VEL
LIN {X 0,Y 512.645,Z 820.335,A -85,B 0,C 180,E1 24765.033,E2 24765.033} C_VEL
LIN {X 0,Y 512.287,Z 830.132,A -85,B 0,C 180,E1 24762.61,E2 24762.61} C_VEL
LIN {X 0,Y 512.085,Z 837.94,A -85,B 0,C 180,E1 24760.233,E2 24760.233} C_VEL
LIN {X 0,Y 511.973,Z 843.91,A -85,B 0,C 180,E1 24757.856,E2 24757.856} C_VEL
LIN {X 0,Y 511.927,Z 848.464,A -85,B 0,C 180,E1 24755.378,E2 24755.378} C_VEL
LIN {X 0,Y 511.914,Z 851.237,A -85,B 0,C 180,E1 24753.022,E2 24753.022} C_VEL
LIN {X 0,Y 511.9,Z 852.373,A -85,B 0,C 180,E1 24750.67,E2 24750.67} C_VEL
LIN {X 0,Y 511.899,Z 852.082,A -85,B 0,C 180,E1 24748.32,E2 24748.32} C_VEL
LIN {X 0,Y 511.91,Z 850.331,A -85,B 0,C 180,E1 24746.079,E2 24746.079} C_VEL
LIN {X 0,Y 511.93,Z 846.807,A -85,B 0,C 180,E1 24743.607,E2 24743.607} C_VEL
LIN {X 0,Y 511.992,Z 841.87,A -85,B 0,C 180,E1 24741.237,E2 24741.237} C_VEL
LIN {X 0,Y 512.127,Z 835.465,A -85,B 0,C 180,E1 24738.969,E2 24738.969} C_VEL
LIN {X 0,Y 512.389,Z 827.051,A -85,B 0,C 180,E1 24736.572,E2 24736.572} C_VEL
LIN {X 0,Y 512.796,Z 817.217,A -85,B 0,C 180,E1 24734.274,E2 24734.274} C_VEL
LIN {X 0,Y 513.345,Z 805.913,A -85,B 0,C 180,E1 24732.076,E2 24732.076} C_VEL
LIN {X 0,Y 514.107,Z 792.55,A -85,B 0,C 180,E1 24729.864,E2 24729.864} C_VEL
LIN {X 0,Y 515.043,Z 778.153,A -85,B 0,C 180,E1 24727.821,E2 24727.821} C_VEL
LIN {X 0,Y 516.124,Z 762.623,A -85,B 0,C 180,E1 24725.933,E2 24725.933} C_VEL
LIN {X 0,Y 517.293,Z 746.261,A -85,B 0,C 180,E1 24724.221,E2 24724.221} C_VEL
LIN {X 0,Y 518.618,Z 727.849,A -85,B 0,C 180,E1 24722.562,E2 24722.562} C_VEL
LIN {X 0,Y 519.964,Z 709.251,A -85,B 0,C 180,E1 24721.14,E2 24721.14} C_VEL
LIN {X 0,Y 521.188,Z 690.011,A -85,B 0,C 180,E1 24719.907,E2 24719.907} C_VEL
LIN {X 0,Y 522.456,Z 669.332,A -85,B 0,C 180,E1 24718.81,E2 24718.81} C_VEL
LIN {X 0,Y 523.533,Z 648.762,A -85,B 0,C 180,E1 24717.931,E2 24717.931} C_VEL
LIN {X 0,Y 524.405,Z 627.76,A -85,B 0,C 180,E1 24717.251,E2 24717.251} C_VEL
LIN {X 0,Y 525.101,Z 605.536,A -85,B 0,C 180,E1 24716.736,E2 24716.736} C_VEL
LIN {X 0,Y 527.851,Z 391.802,A -85,B 0,C 180,E1 24713.437,E2 24713.437} C_VEL
LIN {X 0,Y 528.471,Z 320.059,A -85,B 0,C 180,E1 24712.334,E2 24712.334} C_VEL
LIN {X 0,Y 524.863,Z 299.821,A -85,B 0,C 180,E1 24711.677,E2 24711.677} C_VEL
LIN {X 0,Y 525.254,Z 279.104,A -85,B 0,C 180,E1 24710.192,E2 24710.192} C_VEL
LIN {X 0,Y 516.988,Z 260.027,A -85,B 0,C 180,E1 24708.125,E2 24708.125} C_VEL
LIN {X 0,Y 512.619,Z 248.883,A -85,B 0,C 180,E1 24706.844,E2 24706.844} C_VEL
LIN {X 0,Y 512.614,Z 248.884,A -85,B 0,C 180,E1 24703.481,E2 24703.481} C_VEL
LIN {X 0,Y 512.579,Z 248.885,A -85,B 0,C 180,E1 24700.123,E2 24700.123} C_VEL
LIN {X 0,Y 512.619,Z 248.885,A -85,B 0,C 180,E1 24696.785,E2 24696.785} C_VEL
LIN {X 0,Y 512.594,Z 248.885,A -85,B 0,C 180,E1 24693.506,E2 24693.506} C_VEL
LIN {X 0,Y 512.573,Z 248.886,A -85,B 0,C 180,E1 24690.088,E2 24690.088} C_VEL
LIN {X 0,Y 512.625,Z 248.883,A -85,B 0,C 180,E1 24686.78,E2 24686.78} C_VEL
LIN {X 0,Y 512.591,Z 249.058,A -85,B 0,C 180,E1 24683.899,E2 24683.899} C_VEL
LIN {X 0,Y 513.846,Z 252.328,A -85,B 0,C 180,E1 24683.72,E2 24683.72} C_VEL
LIN {X 0,Y 515.73,Z 254.847,A -85,B 0,C 180,E1 24683.505,E2 24683.505} C_VEL
LIN {X 0,Y 528.348,Z 275.12,A -85,B 0,C 180,E1 24682.085,E2 24682.085} C_VEL
LIN {X 0,Y 525.393,Z 509.084,A -85,B 0,C 180,E1 24678.489,E2 24678.489} C_VEL
LIN {X 0,Y 524.863,Z 534.532,A -85,B 0,C 180,E1 24678.041,E2 24678.041} C_VEL
LIN {X 0,Y 524.06,Z 557.278,A -85,B 0,C 180,E1 24677.424,E2 24677.424} C_VEL
LIN {X 0,Y 522.974,Z 579.815,A -85,B 0,C 180,E1 24676.581,E2 24676.581} C_VEL
LIN {X 0,Y 521.789,Z 600.889,A -85,B 0,C 180,E1 24675.562,E2 24675.562} C_VEL
LIN {X 0,Y 520.535,Z 620.502,A -85,B 0,C 180,E1 24674.405,E2 24674.405} C_VEL
LIN {X 0,Y 519.212,Z 640.034,A -85,B 0,C 180,E1 24673.022,E2 24673.022} C_VEL
LIN {X 0,Y 517.767,Z 659.697,A -85,B 0,C 180,E1 24671.361,E2 24671.361} C_VEL
LIN {X 0,Y 516.527,Z 677.024,A -85,B 0,C 180,E1 24669.64,E2 24669.64} C_VEL
LIN {X 0,Y 515.351,Z 693.787,A -85,B 0,C 180,E1 24667.695,E2 24667.695} C_VEL
LIN {X 0,Y 514.368,Z 708.576,A -85,B 0,C 180,E1 24665.691,E2 24665.691} C_VEL
LIN {X 0,Y 513.527,Z 722.662,A -85,B 0,C 180,E1 24663.462,E2 24663.462} C_VEL
LIN {X 0,Y 512.909,Z 734.562,A -85,B 0,C 180,E1 24661.23,E2 24661.23} C_VEL
LIN {X 0,Y 512.466,Z 745.078,A -85,B 0,C 180,E1 24658.884,E2 24658.884} C_VEL
LIN {X 0,Y 512.186,Z 753.753,A -85,B 0,C 180,E1 24656.532,E2 24656.532} C_VEL
LIN {X 0,Y 512.026,Z 760.685,A -85,B 0,C 180,E1 24654.174,E2 24654.174} C_VEL
LIN {X 0,Y 511.946,Z 765.992,A -85,B 0,C 180,E1 24651.805,E2 24651.805} C_VEL
LIN {X 0,Y 511.916,Z 769.739,A -85,B 0,C 180,E1 24649.422,E2 24649.422} C_VEL
LIN {X 0,Y 511.907,Z 771.882,A -85,B 0,C 180,E1 24647.021,E2 24647.021} C_VEL
LIN {X 0,Y 511.902,Z 772.453,A -85,B 0,C 180,E1 24644.597,E2 24644.597} C_VEL
LIN {X 0,Y 511.91,Z 771.401,A -85,B 0,C 180,E1 24642.145,E2 24642.145} C_VEL
LIN {X 0,Y 511.913,Z 768.783,A -85,B 0,C 180,E1 24639.777,E2 24639.777} C_VEL
LIN {X 0,Y 511.959,Z 764.289,A -85,B 0,C 180,E1 24637.253,E2 24637.253} C_VEL
LIN {X 0,Y 512.08,Z 758.193,A -85,B 0,C 180,E1 24634.81,E2 24634.81} C_VEL
LIN {X 0,Y 512.286,Z 750.303,A -85,B 0,C 180,E1 24632.388,E2 24632.388} C_VEL
LIN {X 0,Y 512.635,Z 740.704,A -85,B 0,C 180,E1 24629.997,E2 24629.997} C_VEL
LIN {X 0,Y 513.146,Z 729.758,A -85,B 0,C 180,E1 24627.734,E2 24627.734} C_VEL
LIN {X 0,Y 513.859,Z 717.045,A -85,B 0,C 180,E1 24625.516,E2 24625.516} C_VEL
LIN {X 0,Y 514.769,Z 702.344,A -85,B 0,C 180,E1 24623.34,E2 24623.34} C_VEL
LIN {X 0,Y 515.857,Z 686.404,A -85,B 0,C 180,E1 24621.322,E2 24621.322} C_VEL
LIN {X 0,Y 517.133,Z 668.612,A -85,B 0,C 180,E1 24619.399,E2 24619.399} C_VEL
LIN {X 0,Y 518.215,Z 653.864,A -85,B 0,C 180,E1 24618.026,E2 24618.026} C_VEL
LIN {X 0,Y 517.768,Z 647.991,A -85,B 0,C 180,E1 24617.466,E2 24617.466} C_VEL
LIN {X 0,Y 513.408,Z 633.381,A -85,B 0,C 180,E1 24616.008,E2 24616.008} C_VEL
LIN {X 0,Y 512.963,Z 627.096,A -85,B 0,C 180,E1 24615.503,E2 24615.503} C_VEL
LIN {X 0,Y 514.376,Z 607.463,A -85,B 0,C 180,E1 24614.254,E2 24614.254} C_VEL
LIN {X 0,Y 515.722,Z 586.647,A -85,B 0,C 180,E1 24613.167,E2 24613.167} C_VEL
LIN {X 0,Y 516.961,Z 564.038,A -85,B 0,C 180,E1 24612.238,E2 24612.238} C_VEL
LIN {X 0,Y 517.921,Z 541.232,A -85,B 0,C 180,E1 24611.542,E2 24611.542} C_VEL
LIN {X 0,Y 518.606,Z 517.468,A -85,B 0,C 180,E1 24611.062,E2 24611.062} C_VEL
LIN {X 0,Y 521.748,Z 290.006,A -85,B 0,C 180,E1 24607.53,E2 24607.53} C_VEL
LIN {X 0,Y 521.792,Z 277.952,A -85,B 0,C 180,E1 24607.329,E2 24607.329} C_VEL
LIN {X 0,Y 509.812,Z 258.95,A -85,B 0,C 180,E1 24605.938,E2 24605.938} C_VEL
LIN {X 0,Y 506.728,Z 254.243,A -85,B 0,C 180,E1 24605.563,E2 24605.563} C_VEL
LIN {X 0,Y 504.942,Z 251.019,A -85,B 0,C 180,E1 24605.334,E2 24605.334} C_VEL
LIN {X 0,Y 504.709,Z 249.852,A -85,B 0,C 180,E1 24605.269,E2 24605.269} C_VEL
LIN {X 0,Y 504.687,Z 249.869,A -85,B 0,C 180,E1 24601.803,E2 24601.803} C_VEL
LIN {X 0,Y 504.673,Z 249.871,A -85,B 0,C 180,E1 24598.392,E2 24598.392} C_VEL
LIN {X 0,Y 504.708,Z 249.867,A -85,B 0,C 180,E1 24594.96,E2 24594.96} C_VEL
LIN {X 0,Y 504.694,Z 249.867,A -85,B 0,C 180,E1 24591.501,E2 24591.501} C_VEL
LIN {X 0,Y 504.666,Z 249.869,A -85,B 0,C 180,E1 24588.004,E2 24588.004} C_VEL
LIN {X 0,Y 504.689,Z 249.868,A -85,B 0,C 180,E1 24584.573,E2 24584.573} C_VEL
LIN {X 0,Y 504.707,Z 249.865,A -85,B 0,C 180,E1 24581.08,E2 24581.08} C_VEL
LIN {X 0,Y 504.667,Z 249.866,A -85,B 0,C 180,E1 24577.629,E2 24577.629} C_VEL
LIN {X 0,Y 504.666,Z 249.868,A -85,B 0,C 180,E1 24574.091,E2 24574.091} C_VEL
LIN {X 0,Y 504.71,Z 249.867,A -85,B 0,C 180,E1 24570.682,E2 24570.682} C_VEL
LIN {X 0,Y 504.676,Z 249.865,A -85,B 0,C 180,E1 24567.276,E2 24567.276} C_VEL
LIN {X 0,Y 504.659,Z 249.868,A -85,B 0,C 180,E1 24563.86,E2 24563.86} C_VEL
LIN {X 0,Y 504.705,Z 249.867,A -85,B 0,C 180,E1 24560.537,E2 24560.537} C_VEL
LIN {X 0,Y 504.677,Z 249.865,A -85,B 0,C 180,E1 24557.065,E2 24557.065} C_VEL
LIN {X 0,Y 504.653,Z 249.868,A -85,B 0,C 180,E1 24553.661,E2 24553.661} C_VEL
LIN {X 0,Y 504.689,Z 249.867,A -85,B 0,C 180,E1 24550.219,E2 24550.219} C_VEL
LIN {X 0,Y 504.684,Z 249.867,A -85,B 0,C 180,E1 24546.81,E2 24546.81} C_VEL
LIN {X 0,Y 504.65,Z 249.869,A -85,B 0,C 180,E1 24543.401,E2 24543.401} C_VEL
LIN {X 0,Y 504.677,Z 249.872,A -85,B 0,C 180,E1 24539.966,E2 24539.966} C_VEL
LIN {X 0,Y 504.689,Z 249.864,A -85,B 0,C 180,E1 24536.583,E2 24536.583} C_VEL
LIN {X 0,Y 504.646,Z 249.866,A -85,B 0,C 180,E1 24533.168,E2 24533.168} C_VEL
LIN {X 0,Y 504.664,Z 249.87,A -85,B 0,C 180,E1 24529.706,E2 24529.706} C_VEL
LIN {X 0,Y 504.698,Z 249.87,A -85,B 0,C 180,E1 24526.308,E2 24526.308} C_VEL
LIN {X 0,Y 504.643,Z 249.87,A -85,B 0,C 180,E1 24522.963,E2 24522.963} C_VEL
LIN {X 0,Y 504.647,Z 249.868,A -85,B 0,C 180,E1 24519.405,E2 24519.405} C_VEL
LIN {X 0,Y 504.701,Z 249.871,A -85,B 0,C 180,E1 24516.04,E2 24516.04} C_VEL
LIN {X 0,Y 504.647,Z 249.871,A -85,B 0,C 180,E1 24512.607,E2 24512.607} C_VEL
LIN {X 0,Y 504.639,Z 249.87,A -85,B 0,C 180,E1 24509.104,E2 24509.104} C_VEL
LIN {X 0,Y 504.695,Z 249.866,A -85,B 0,C 180,E1 24505.837,E2 24505.837} C_VEL
LIN {X 0,Y 504.642,Z 249.871,A -85,B 0,C 180,E1 24502.48,E2 24502.48} C_VEL
LIN {X 0,Y 504.633,Z 249.871,A -85,B 0,C 180,E1 24498.96,E2 24498.96} C_VEL
LIN {X 0,Y 504.692,Z 249.871,A -85,B 0,C 180,E1 24495.629,E2 24495.629} C_VEL
LIN {X 0,Y 504.642,Z 249.872,A -85,B 0,C 180,E1 24492.238,E2 24492.238} C_VEL
LIN {X 0,Y 504.628,Z 249.873,A -85,B 0,C 180,E1 24488.774,E2 24488.774} C_VEL
LIN {X 0,Y 504.681,Z 249.872,A -85,B 0,C 180,E1 24485.455,E2 24485.455} C_VEL
LIN {X 0,Y 504.644,Z 249.873,A -85,B 0,C 180,E1 24482.042,E2 24482.042} C_VEL
LIN {X 0,Y 504.628,Z 249.872,A -85,B 0,C 180,E1 24478.636,E2 24478.636} C_VEL
LIN {X 0,Y 504.675,Z 249.869,A -85,B 0,C 180,E1 24475.225,E2 24475.225} C_VEL
LIN {X 0,Y 504.647,Z 249.872,A -85,B 0,C 180,E1 24471.912,E2 24471.912} C_VEL
LIN {X 0,Y 504.632,Z 249.87,A -85,B 0,C 180,E1 24468.455,E2 24468.455} C_VEL
LIN {X 0,Y 504.68,Z 249.87,A -85,B 0,C 180,E1 24465.074,E2 24465.074} C_VEL
LIN {X 0,Y 504.652,Z 249.872,A -85,B 0,C 180,E1 24461.756,E2 24461.756} C_VEL
LIN {X 0,Y 504.636,Z 249.87,A -85,B 0,C 180,E1 24458.313,E2 24458.313} C_VEL
LIN {X 0,Y 504.694,Z 249.867,A -85,B 0,C 180,E1 24455.039,E2 24455.039} C_VEL
LIN {X 0,Y 504.658,Z 249.87,A -85,B 0,C 180,E1 24451.607,E2 24451.607} C_VEL
LIN {X 0,Y 504.642,Z 249.872,A -85,B 0,C 180,E1 24448.194,E2 24448.194} C_VEL
LIN {X 0,Y 504.69,Z 249.871,A -85,B 0,C 180,E1 24444.794,E2 24444.794} C_VEL
LIN {X 0,Y 504.669,Z 249.872,A -85,B 0,C 180,E1 24441.384,E2 24441.384} C_VEL
LIN {X 0,Y 504.646,Z 249.875,A -85,B 0,C 180,E1 24437.957,E2 24437.957} C_VEL
LIN {X 0,Y 504.679,Z 249.874,A -85,B 0,C 180,E1 24434.501,E2 24434.501} C_VEL
LIN {X 0,Y 504.706,Z 250.136,A -85,B 0,C 180,E1 24434.39,E2 24434.39} C_VEL
LIN {X 0,Y 505.899,Z 253.277,A -85,B 0,C 180,E1 24433.994,E2 24433.994} C_VEL
LIN {X 0,Y 511.759,Z 266.262,A -85,B 0,C 180,E1 24432.31,E2 24432.31} C_VEL
LIN {X 0,Y 519.328,Z 283.788,A -85,B 0,C 180,E1 24430.189,E2 24430.189} C_VEL
LIN {X 0,Y 518.601,Z 301.987,A -85,B 0,C 180,E1 24428.839,E2 24428.839} C_VEL
LIN {X 0,Y 522.302,Z 323.558,A -85,B 0,C 180,E1 24428.138,E2 24428.138} C_VEL
LIN {X 0,Y 519.317,Z 543.814,A -85,B 0,C 180,E1 24424.722,E2 24424.722} C_VEL
LIN {X 0,Y 518.34,Z 609.626,A -85,B 0,C 180,E1 24423.676,E2 24423.676} C_VEL
LIN {X 0,Y 517.513,Z 630.952,A -85,B 0,C 180,E1 24423.14,E2 24423.14} C_VEL
LIN {X 0,Y 516.464,Z 653.244,A -85,B 0,C 180,E1 24422.362,E2 24422.362} C_VEL
LIN {X 0,Y 515.306,Z 673.409,A -85,B 0,C 180,E1 24421.461,E2 24421.461} C_VEL
LIN {X 0,Y 513.904,Z 693.777,A -85,B 0,C 180,E1 24420.322,E2 24420.322} C_VEL
LIN {X 0,Y 512.479,Z 713.33,A -85,B 0,C 180,E1 24419,E2 24419} C_VEL
LIN {X 0,Y 511.085,Z 731.442,A -85,B 0,C 180,E1 24417.558,E2 24417.558} C_VEL
LIN {X 0,Y 509.65,Z 749.309,A -85,B 0,C 180,E1 24415.881,E2 24415.881} C_VEL
LIN {X 0,Y 508.387,Z 765.238,A -85,B 0,C 180,E1 24414.138,E2 24414.138} C_VEL
LIN {X 0,Y 507.247,Z 780.335,A -85,B 0,C 180,E1 24412.237,E2 24412.237} C_VEL
LIN {X 0,Y 506.224,Z 794.875,A -85,B 0,C 180,E1 24410.099,E2 24410.099} C_VEL
LIN {X 0,Y 505.418,Z 807.549,A -85,B 0,C 180,E1 24407.907,E2 24407.907} C_VEL
LIN {X 0,Y 504.787,Z 819.305,A -85,B 0,C 180,E1 24405.508,E2 24405.508} C_VEL
LIN {X 0,Y 504.382,Z 828.854,A -85,B 0,C 180,E1 24403.176,E2 24403.176} C_VEL
LIN {X 0,Y 504.128,Z 836.533,A -85,B 0,C 180,E1 24400.859,E2 24400.859} C_VEL
LIN {X 0,Y 503.994,Z 843.148,A -85,B 0,C 180,E1 24398.326,E2 24398.326} C_VEL
LIN {X 0,Y 503.931,Z 847.825,A -85,B 0,C 180,E1 24395.921,E2 24395.921} C_VEL
LIN {X 0,Y 503.909,Z 850.788,A -85,B 0,C 180,E1 24393.525,E2 24393.525} C_VEL
LIN {X 0,Y 503.912,Z 852.305,A -85,B 0,C 180,E1 24391.022,E2 24391.022} C_VEL
LIN {X 0,Y 503.909,Z 852.259,A -85,B 0,C 180,E1 24388.748,E2 24388.748} C_VEL
LIN {X 0,Y 503.908,Z 850.671,A -85,B 0,C 180,E1 24386.358,E2 24386.358} C_VEL
LIN {X 0,Y 503.933,Z 847.63,A -85,B 0,C 180,E1 24383.963,E2 24383.963} C_VEL
LIN {X 0,Y 503.992,Z 842.888,A -85,B 0,C 180,E1 24381.557,E2 24381.557} C_VEL
LIN {X 0,Y 504.137,Z 836.172,A -85,B 0,C 180,E1 24379.023,E2 24379.023} C_VEL
LIN {X 0,Y 504.4,Z 828.424,A -85,B 0,C 180,E1 24376.705,E2 24376.705} C_VEL
LIN {X 0,Y 504.819,Z 818.776,A -85,B 0,C 180,E1 24374.373,E2 24374.373} C_VEL
LIN {X 0,Y 505.442,Z 807.181,A -85,B 0,C 180,E1 24372.024,E2 24372.024} C_VEL
LIN {X 0,Y 506.225,Z 794.859,A -85,B 0,C 180,E1 24369.898,E2 24369.898} C_VEL
LIN {X 0,Y 507.249,Z 780.319,A -85,B 0,C 180,E1 24367.761,E2 24367.761} C_VEL
LIN {X 0,Y 508.434,Z 764.649,A -85,B 0,C 180,E1 24365.793,E2 24365.793} C_VEL
LIN {X 0,Y 509.84,Z 746.928,A -85,B 0,C 180,E1 24363.884,E2 24363.884} C_VEL
LIN {X 0,Y 511.24,Z 729.305,A -85,B 0,C 180,E1 24362.259,E2 24362.259} C_VEL
LIN {X 0,Y 512.681,Z 710.87,A -85,B 0,C 180,E1 24360.819,E2 24360.819} C_VEL
LIN {X 0,Y 514.039,Z 691.732,A -85,B 0,C 180,E1 24359.555,E2 24359.555} C_VEL
LIN {X 0,Y 515.386,Z 672.142,A -85,B 0,C 180,E1 24358.477,E2 24358.477} C_VEL
LIN {X 0,Y 516.543,Z 651.718,A -85,B 0,C 180,E1 24357.575,E2 24357.575} C_VEL
LIN {X 0,Y 517.566,Z 629.896,A -85,B 0,C 180,E1 24356.83,E2 24356.83} C_VEL
LIN {X 0,Y 518.363,Z 608.585,A -85,B 0,C 180,E1 24356.305,E2 24356.305} C_VEL
LIN {X 0,Y 520.005,Z 490.844,A -85,B 0,C 180,E1 24354.464,E2 24354.464} C_VEL
LIN {X 0,Y 521.915,Z 321.871,A -85,B 0,C 180,E1 24351.871,E2 24351.871} C_VEL
LIN {X 0,Y 517.838,Z 298.188,A -85,B 0,C 180,E1 24351.09,E2 24351.09} C_VEL
LIN {X 0,Y 518.131,Z 282.22,A -85,B 0,C 180,E1 24349.92,E2 24349.92} C_VEL
LIN {X 0,Y 510.482,Z 264.349,A -85,B 0,C 180,E1 24347.931,E2 24347.931} C_VEL
LIN {X 0,Y 506.112,Z 253.564,A -85,B 0,C 180,E1 24346.637,E2 24346.637} C_VEL
LIN {X 0,Y 504.656,Z 249.957,A -85,B 0,C 180,E1 24346.18,E2 24346.18} C_VEL
LIN {X 0,Y 504.68,Z 249.874,A -85,B 0,C 180,E1 24342.809,E2 24342.809} C_VEL
LIN {X 0,Y 504.667,Z 249.873,A -85,B 0,C 180,E1 24339.493,E2 24339.493} C_VEL
LIN {X 0,Y 504.638,Z 249.874,A -85,B 0,C 180,E1 24336.048,E2 24336.048} C_VEL
LIN {X 0,Y 504.665,Z 249.874,A -85,B 0,C 180,E1 24332.609,E2 24332.609} C_VEL
LIN {X 0,Y 504.666,Z 249.873,A -85,B 0,C 180,E1 24329.3,E2 24329.3} C_VEL
LIN {X 0,Y 504.631,Z 249.877,A -85,B 0,C 180,E1 24325.901,E2 24325.901} C_VEL
LIN {X 0,Y 504.688,Z 249.996,A -85,B 0,C 180,E1 24324.63,E2 24324.63} C_VEL
LIN {X 0,Y 505.995,Z 253.413,A -85,B 0,C 180,E1 24324.431,E2 24324.431} C_VEL
LIN {X 0,Y 507.832,Z 255.896,A -85,B 0,C 180,E1 24324.204,E2 24324.204} C_VEL
LIN {X 0,Y 521.016,Z 276.753,A -85,B 0,C 180,E1 24322.656,E2 24322.656} C_VEL
LIN {X 0,Y 521.862,Z 278.676,A -85,B 0,C 180,E1 24322.554,E2 24322.554} C_VEL
LIN {X 0,Y 519.914,Z 419.683,A -85,B 0,C 180,E1 24320.357,E2 24320.357} C_VEL
LIN {X 0,Y 518.353,Z 528.371,A -85,B 0,C 180,E1 24318.654,E2 24318.654} C_VEL
LIN {X 0,Y 517.58,Z 550.191,A -85,B 0,C 180,E1 24318.122,E2 24318.122} C_VEL
LIN {X 0,Y 516.514,Z 572.726,A -85,B 0,C 180,E1 24317.345,E2 24317.345} C_VEL
LIN {X 0,Y 515.211,Z 594.816,A -85,B 0,C 180,E1 24316.345,E2 24316.345} C_VEL
LIN {X 0,Y 513.798,Z 615.476,A -85,B 0,C 180,E1 24315.174,E2 24315.174} C_VEL
LIN {X 0,Y 512.357,Z 635.05,A -85,B 0,C 180,E1 24313.832,E2 24313.832} C_VEL
LIN {X 0,Y 510.865,Z 654.323,A -85,B 0,C 180,E1 24312.262,E2 24312.262} C_VEL
LIN {X 0,Y 509.403,Z 672.41,A -85,B 0,C 180,E1 24310.519,E2 24310.519} C_VEL
LIN {X 0,Y 508.076,Z 689.412,A -85,B 0,C 180,E1 24308.603,E2 24308.603} C_VEL
LIN {X 0,Y 506.868,Z 705.592,A -85,B 0,C 180,E1 24306.457,E2 24306.457} C_VEL
LIN {X 0,Y 505.925,Z 719.428,A -85,B 0,C 180,E1 24304.308,E2 24304.308} C_VEL
LIN {X 0,Y 505.156,Z 732.413,A -85,B 0,C 180,E1 24301.93,E2 24301.93} C_VEL
LIN {X 0,Y 504.616,Z 743.287,A -85,B 0,C 180,E1 24299.547,E2 24299.547} C_VEL
LIN {X 0,Y 504.263,Z 752.283,A -85,B 0,C 180,E1 24297.16,E2 24297.16} C_VEL
LIN {X 0,Y 504.06,Z 759.6,A -85,B 0,C 180,E1 24294.733,E2 24294.733} C_VEL
LIN {X 0,Y 503.954,Z 765.389,A -85,B 0,C 180,E1 24292.248,E2 24292.248} C_VEL
LIN {X 0,Y 503.911,Z 769.37,A -85,B 0,C 180,E1 24289.791,E2 24289.791} C_VEL
LIN {X 0,Y 503.911,Z 771.753,A -85,B 0,C 180,E1 24287.278,E2 24287.278} C_VEL
LIN {X 0,Y 503.91,Z 772.484,A -85,B 0,C 180,E1 24284.818,E2 24284.818} C_VEL
LIN {X 0,Y 503.909,Z 771.558,A -85,B 0,C 180,E1 24282.329,E2 24282.329} C_VEL
LIN {X 0,Y 503.914,Z 768.94,A -85,B 0,C 180,E1 24279.805,E2 24279.805} C_VEL
LIN {X 0,Y 503.959,Z 764.651,A -85,B 0,C 180,E1 24277.305,E2 24277.305} C_VEL
LIN {X 0,Y 504.082,Z 758.826,A -85,B 0,C 180,E1 24274.885,E2 24274.885} C_VEL
LIN {X 0,Y 504.301,Z 751.371,A -85,B 0,C 180,E1 24272.489,E2 24272.489} C_VEL
LIN {X 0,Y 504.689,Z 741.651,A -85,B 0,C 180,E1 24269.97,E2 24269.97} C_VEL
LIN {X 0,Y 505.262,Z 730.345,A -85,B 0,C 180,E1 24267.572,E2 24267.572} C_VEL
LIN {X 0,Y 506.06,Z 717.488,A -85,B 0,C 180,E1 24265.278,E2 24265.278} C_VEL
LIN {X 0,Y 507.054,Z 703.044,A -85,B 0,C 180,E1 24263.095,E2 24263.095} C_VEL
LIN {X 0,Y 508.239,Z 687.346,A -85,B 0,C 180,E1 24261.06,E2 24261.06} C_VEL
LIN {X 0,Y 509.605,Z 669.923,A -85,B 0,C 180,E1 24259.134,E2 24259.134} C_VEL
LIN {X 0,Y 511.016,Z 652.39,A -85,B 0,C 180,E1 24257.479,E2 24257.479} C_VEL
LIN {X 0,Y 512.59,Z 632.208,A -85,B 0,C 180,E1 24255.867,E2 24255.867} C_VEL
LIN {X 0,Y 512.963,Z 627.096,A -85,B 0,C 180,E1 24255.503,E2 24255.503} C_VEL
LIN {X 0,Y 512.546,Z 620.707,A -85,B 0,C 180,E1 24255.011,E2 24255.011} C_VEL
LIN {X 0,Y 508.425,Z 604.895,A -85,B 0,C 180,E1 24253.694,E2 24253.694} C_VEL
LIN {X 0,Y 508.055,Z 598.161,A -85,B 0,C 180,E1 24253.265,E2 24253.265} C_VEL
LIN {X 0,Y 509.432,Z 577.475,A -85,B 0,C 180,E1 24252.278,E2 24252.278} C_VEL
LIN {X 0,Y 510.602,Z 555.358,A -85,B 0,C 180,E1 24251.453,E2 24251.453} C_VEL
LIN {X 0,Y 511.551,Z 532.735,A -85,B 0,C 180,E1 24250.849,E2 24250.849} C_VEL
LIN {X 0,Y 512.193,Z 498.303,A -85,B 0,C 180,E1 24250.273,E2 24250.273} C_VEL
LIN {X 0,Y 515.401,Z 288.152,A -85,B 0,C 180,E1 24246.962,E2 24246.962} C_VEL
LIN {X 0,Y 515.35,Z 281.056,A -85,B 0,C 180,E1 24246.835,E2 24246.835} C_VEL
LIN {X 0,Y 504.288,Z 263.656,A -85,B 0,C 180,E1 24245.517,E2 24245.517} C_VEL
LIN {X 0,Y 499.215,Z 255.691,A -85,B 0,C 180,E1 24244.878,E2 24244.878} C_VEL
LIN {X 0,Y 497.185,Z 252.67,A -85,B 0,C 180,E1 24244.62,E2 24244.62} C_VEL
LIN {X 0,Y 496.737,Z 250.861,A -85,B 0,C 180,E1 24244.516,E2 24244.516} C_VEL
LIN {X 0,Y 496.77,Z 250.859,A -85,B 0,C 180,E1 24240.978,E2 24240.978} C_VEL
LIN {X 0,Y 496.772,Z 250.856,A -85,B 0,C 180,E1 24237.432,E2 24237.432} C_VEL
LIN {X 0,Y 496.733,Z 250.858,A -85,B 0,C 180,E1 24233.965,E2 24233.965} C_VEL
LIN {X 0,Y 496.735,Z 250.86,A -85,B 0,C 180,E1 24230.38,E2 24230.38} C_VEL
LIN {X 0,Y 496.77,Z 250.856,A -85,B 0,C 180,E1 24226.849,E2 24226.849} C_VEL
LIN {X 0,Y 496.753,Z 250.852,A -85,B 0,C 180,E1 24223.385,E2 24223.385} C_VEL
LIN {X 0,Y 496.726,Z 250.857,A -85,B 0,C 180,E1 24219.853,E2 24219.853} C_VEL
LIN {X 0,Y 496.74,Z 250.856,A -85,B 0,C 180,E1 24216.357,E2 24216.357} C_VEL
LIN {X 0,Y 496.77,Z 250.855,A -85,B 0,C 180,E1 24212.885,E2 24212.885} C_VEL
LIN {X 0,Y 496.731,Z 250.852,A -85,B 0,C 180,E1 24209.424,E2 24209.424} C_VEL
LIN {X 0,Y 496.719,Z 250.851,A -85,B 0,C 180,E1 24205.846,E2 24205.846} C_VEL
LIN {X 0,Y 496.753,Z 250.853,A -85,B 0,C 180,E1 24202.367,E2 24202.367} C_VEL
LIN {X 0,Y 496.759,Z 250.854,A -85,B 0,C 180,E1 24198.86,E2 24198.86} C_VEL
LIN {X 0,Y 496.717,Z 250.856,A -85,B 0,C 180,E1 24195.428,E2 24195.428} C_VEL
LIN {X 0,Y 496.722,Z 250.858,A -85,B 0,C 180,E1 24191.813,E2 24191.813} C_VEL
LIN {X 0,Y 496.77,Z 250.857,A -85,B 0,C 180,E1 24188.389,E2 24188.389} C_VEL
LIN {X 0,Y 496.733,Z 250.854,A -85,B 0,C 180,E1 24184.923,E2 24184.923} C_VEL
LIN {X 0,Y 496.712,Z 250.856,A -85,B 0,C 180,E1 24181.508,E2 24181.508} C_VEL
LIN {X 0,Y 496.754,Z 250.856,A -85,B 0,C 180,E1 24178.141,E2 24178.141} C_VEL
LIN {X 0,Y 496.734,Z 250.859,A -85,B 0,C 180,E1 24174.714,E2 24174.714} C_VEL
LIN {X 0,Y 496.706,Z 250.861,A -85,B 0,C 180,E1 24171.244,E2 24171.244} C_VEL
LIN {X 0,Y 496.73,Z 250.861,A -85,B 0,C 180,E1 24167.757,E2 24167.757} C_VEL
LIN {X 0,Y 496.755,Z 250.858,A -85,B 0,C 180,E1 24164.298,E2 24164.298} C_VEL
LIN {X 0,Y 496.706,Z 250.861,A -85,B 0,C 180,E1 24160.857,E2 24160.857} C_VEL
LIN {X 0,Y 496.706,Z 250.861,A -85,B 0,C 180,E1 24157.291,E2 24157.291} C_VEL
LIN {X 0,Y 496.757,Z 250.857,A -85,B 0,C 180,E1 24153.883,E2 24153.883} C_VEL
LIN {X 0,Y 496.716,Z 250.857,A -85,B 0,C 180,E1 24150.479,E2 24150.479} C_VEL
LIN {X 0,Y 496.698,Z 250.859,A -85,B 0,C 180,E1 24147.059,E2 24147.059} C_VEL
LIN {X 0,Y 496.739,Z 250.861,A -85,B 0,C 180,E1 24143.611,E2 24143.611} C_VEL
LIN {X 0,Y 496.716,Z 250.858,A -85,B 0,C 180,E1 24140.254,E2 24140.254} C_VEL
LIN {X 0,Y 496.693,Z 250.86,A -85,B 0,C 180,E1 24136.849,E2 24136.849} C_VEL
LIN {X 0,Y 496.739,Z 250.861,A -85,B 0,C 180,E1 24133.501,E2 24133.501} C_VEL
LIN {X 0,Y 496.713,Z 250.858,A -85,B 0,C 180,E1 24130.084,E2 24130.084} C_VEL
LIN {X 0,Y 496.687,Z 250.86,A -85,B 0,C 180,E1 24126.703,E2 24126.703} C_VEL
LIN {X 0,Y 496.726,Z 250.862,A -85,B 0,C 180,E1 24123.278,E2 24123.278} C_VEL
LIN {X 0,Y 496.716,Z 250.858,A -85,B 0,C 180,E1 24119.883,E2 24119.883} C_VEL
LIN {X 0,Y 496.689,Z 250.861,A -85,B 0,C 180,E1 24116.421,E2 24116.421} C_VEL
LIN {X 0,Y 496.712,Z 250.861,A -85,B 0,C 180,E1 24112.945,E2 24112.945} C_VEL
LIN {X 0,Y 496.741,Z 250.862,A -85,B 0,C 180,E1 24109.562,E2 24109.562} C_VEL
LIN {X 0,Y 496.696,Z 250.859,A -85,B 0,C 180,E1 24106.139,E2 24106.139} C_VEL
LIN {X 0,Y 496.701,Z 250.86,A -85,B 0,C 180,E1 24102.545,E2 24102.545} C_VEL
LIN {X 0,Y 496.759,Z 250.855,A -85,B 0,C 180,E1 24099.128,E2 24099.128} C_VEL
LIN {X 0,Y 496.711,Z 250.859,A -85,B 0,C 180,E1 24095.754,E2 24095.754} C_VEL
LIN {X 0,Y 496.704,Z 250.858,A -85,B 0,C 180,E1 24092.289,E2 24092.289} C_VEL
LIN {X 0,Y 496.763,Z 250.857,A -85,B 0,C 180,E1 24088.984,E2 24088.984} C_VEL
LIN {X 0,Y 496.719,Z 250.863,A -85,B 0,C 180,E1 24085.553,E2 24085.553} C_VEL
LIN {X 0,Y 496.706,Z 250.86,A -85,B 0,C 180,E1 24082.097,E2 24082.097} C_VEL
LIN {X 0,Y 496.751,Z 250.861,A -85,B 0,C 180,E1 24078.684,E2 24078.684} C_VEL
LIN {X 0,Y 496.743,Z 250.863,A -85,B 0,C 180,E1 24075.183,E2 24075.183} C_VEL
LIN {X 0,Y 498.065,Z 254.345,A -85,B 0,C 180,E1 24074.711,E2 24074.711} C_VEL
LIN {X 0,Y 505.445,Z 270.758,A -85,B 0,C 180,E1 24072.534,E2 24072.534} C_VEL
LIN {X 0,Y 512.532,Z 287.165,A -85,B 0,C 180,E1 24070.511,E2 24070.511} C_VEL
LIN {X 0,Y 511.943,Z 301.548,A -85,B 0,C 180,E1 24069.437,E2 24069.437} C_VEL
LIN {X 0,Y 515.891,Z 325.024,A -85,B 0,C 180,E1 24068.65,E2 24068.65} C_VEL
LIN {X 0,Y 512.637,Z 541.982,A -85,B 0,C 180,E1 24065.238,E2 24065.238} C_VEL
LIN {X 0,Y 511.645,Z 609.852,A -85,B 0,C 180,E1 24064.164,E2 24064.164} C_VEL
LIN {X 0,Y 510.832,Z 630.246,A -85,B 0,C 180,E1 24063.653,E2 24063.653} C_VEL
LIN {X 0,Y 509.698,Z 652.426,A -85,B 0,C 180,E1 24062.882,E2 24062.882} C_VEL
LIN {X 0,Y 508.49,Z 672.195,A -85,B 0,C 180,E1 24061.999,E2 24061.999} C_VEL
LIN {X 0,Y 507.033,Z 691.765,A -85,B 0,C 180,E1 24060.909,E2 24060.909} C_VEL
LIN {X 0,Y 505.412,Z 712.515,A -85,B 0,C 180,E1 24059.51,E2 24059.51} C_VEL
LIN {X 0,Y 503.87,Z 730.77,A -85,B 0,C 180,E1 24058.052,E2 24058.052} C_VEL
LIN {X 0,Y 502.309,Z 748.716,A -85,B 0,C 180,E1 24056.35,E2 24056.35} C_VEL
LIN {X 0,Y 500.871,Z 765.174,A -85,B 0,C 180,E1 24054.531,E2 24054.531} C_VEL
LIN {X 0,Y 499.612,Z 780.336,A -85,B 0,C 180,E1 24052.595,E2 24052.595} C_VEL
LIN {X 0,Y 498.484,Z 794.874,A -85,B 0,C 180,E1 24050.425,E2 24050.425} C_VEL
LIN {X 0,Y 497.624,Z 807.192,A -85,B 0,C 180,E1 24048.266,E2 24048.266} C_VEL
LIN {X 0,Y 496.931,Z 818.788,A -85,B 0,C 180,E1 24045.88,E2 24045.88} C_VEL
LIN {X 0,Y 496.464,Z 828.435,A -85,B 0,C 180,E1 24043.509,E2 24043.509} C_VEL
LIN {X 0,Y 496.158,Z 836.441,A -85,B 0,C 180,E1 24041.066,E2 24041.066} C_VEL
LIN {X 0,Y 495.996,Z 842.894,A -85,B 0,C 180,E1 24038.578,E2 24038.578} C_VEL
LIN {X 0,Y 495.936,Z 847.638,A -85,B 0,C 180,E1 24036.133,E2 24036.133} C_VEL
LIN {X 0,Y 495.907,Z 850.675,A -85,B 0,C 180,E1 24033.698,E2 24033.698} C_VEL
LIN {X 0,Y 495.91,Z 852.282,A -85,B 0,C 180,E1 24031.154,E2 24031.154} C_VEL
LIN {X 0,Y 495.91,Z 852.281,A -85,B 0,C 180,E1 24028.844,E2 24028.844} C_VEL
LIN {X 0,Y 495.908,Z 850.671,A -85,B 0,C 180,E1 24026.3,E2 24026.3} C_VEL
LIN {X 0,Y 495.937,Z 847.63,A -85,B 0,C 180,E1 24023.865,E2 24023.865} C_VEL
LIN {X 0,Y 495.998,Z 843.142,A -85,B 0,C 180,E1 24021.537,E2 24021.537} C_VEL
LIN {X 0,Y 496.148,Z 836.878,A -85,B 0,C 180,E1 24019.079,E2 24019.079} C_VEL
LIN {X 0,Y 496.423,Z 829.253,A -85,B 0,C 180,E1 24016.725,E2 24016.725} C_VEL
LIN {X 0,Y 496.868,Z 819.807,A -85,B 0,C 180,E1 24014.356,E2 24014.356} C_VEL
LIN {X 0,Y 497.539,Z 808.449,A -85,B 0,C 180,E1 24011.971,E2 24011.971} C_VEL
LIN {X 0,Y 498.434,Z 795.624,A -85,B 0,C 180,E1 24009.693,E2 24009.693} C_VEL
LIN {X 0,Y 499.541,Z 781.17,A -85,B 0,C 180,E1 24007.523,E2 24007.523} C_VEL
LIN {X 0,Y 500.806,Z 765.952,A -85,B 0,C 180,E1 24005.562,E2 24005.562} C_VEL
LIN {X 0,Y 502.26,Z 749.298,A -85,B 0,C 180,E1 24003.708,E2 24003.708} C_VEL
LIN {X 0,Y 503.79,Z 731.659,A -85,B 0,C 180,E1 24002.029,E2 24002.029} C_VEL
LIN {X 0,Y 505.353,Z 713.219,A -85,B 0,C 180,E1 24000.542,E2 24000.542} C_VEL
LIN {X 0,Y 506.89,Z 693.738,A -85,B 0,C 180,E1 23999.211,E2 23999.211} C_VEL
LIN {X 0,Y 508.412,Z 673.363,A -85,B 0,C 180,E1 23998.06,E2 23998.06} C_VEL
LIN {X 0,Y 509.657,Z 653.194,A -85,B 0,C 180,E1 23997.149,E2 23997.149} C_VEL
LIN {X 0,Y 510.815,Z 630.755,A -85,B 0,C 180,E1 23996.362,E2 23996.362} C_VEL
LIN {X 0,Y 511.618,Z 610.589,A -85,B 0,C 180,E1 23995.853,E2 23995.853} C_VEL
LIN {X 0,Y 512.157,Z 571.995,A -85,B 0,C 180,E1 23995.239,E2 23995.239} C_VEL
LIN {X 0,Y 514.034,Z 419.788,A -85,B 0,C 180,E1 23992.917,E2 23992.917} C_VEL
LIN {X 0,Y 515.36,Z 323.148,A -85,B 0,C 180,E1 23991.366,E2 23991.366} C_VEL
LIN {X 0,Y 510.893,Z 296.154,A -85,B 0,C 180,E1 23990.452,E2 23990.452} C_VEL
LIN {X 0,Y 511.013,Z 285.366,A -85,B 0,C 180,E1 23989.635,E2 23989.635} C_VEL
LIN {X 0,Y 504.014,Z 268.705,A -85,B 0,C 180,E1 23987.728,E2 23987.728} C_VEL
LIN {X 0,Y 499.717,Z 258.116,A -85,B 0,C 180,E1 23986.412,E2 23986.412} C_VEL
LIN {X 0,Y 496.875,Z 251.654,A -85,B 0,C 180,E1 23985.526,E2 23985.526} C_VEL
LIN {X 0,Y 496.747,Z 250.862,A -85,B 0,C 180,E1 23985.413,E2 23985.413} C_VEL
LIN {X 0,Y 496.705,Z 250.864,A -85,B 0,C 180,E1 23982.029,E2 23982.029} C_VEL
LIN {X 0,Y 496.723,Z 250.864,A -85,B 0,C 180,E1 23978.61,E2 23978.61} C_VEL
LIN {X 0,Y 496.755,Z 250.86,A -85,B 0,C 180,E1 23975.146,E2 23975.146} C_VEL
LIN {X 0,Y 496.698,Z 250.864,A -85,B 0,C 180,E1 23971.831,E2 23971.831} C_VEL
LIN {X 0,Y 496.709,Z 250.865,A -85,B 0,C 180,E1 23968.364,E2 23968.364} C_VEL
LIN {X 0,Y 496.741,Z 251.104,A -85,B 0,C 180,E1 23965.435,E2 23965.435} C_VEL
LIN {X 0,Y 498.047,Z 254.369,A -85,B 0,C 180,E1 23965.222,E2 23965.222} C_VEL
LIN {X 0,Y 500.108,Z 256.95,A -85,B 0,C 180,E1 23964.952,E2 23964.952} C_VEL
LIN {X 0,Y 510.999,Z 274.323,A -85,B 0,C 180,E1 23963.55,E2 23963.55} C_VEL
LIN {X 0,Y 515.357,Z 281.694,A -85,B 0,C 180,E1 23963.033,E2 23963.033} C_VEL
LIN {X 0,Y 513.023,Z 427.935,A -85,B 0,C 180,E1 23960.702,E2 23960.702} C_VEL
LIN {X 0,Y 511.649,Z 528.841,A -85,B 0,C 180,E1 23959.137,E2 23959.137} C_VEL
LIN {X 0,Y 510.888,Z 549.822,A -85,B 0,C 180,E1 23958.626,E2 23958.626} C_VEL
LIN {X 0,Y 509.694,Z 573.003,A -85,B 0,C 180,E1 23957.821,E2 23957.821} C_VEL
LIN {X 0,Y 508.29,Z 595.05,A -85,B 0,C 180,E1 23956.809,E2 23956.809} C_VEL
LIN {X 0,Y 506.75,Z 615.687,A -85,B 0,C 180,E1 23955.625,E2 23955.625} C_VEL
LIN {X 0,Y 505.196,Z 635.209,A -85,B 0,C 180,E1 23954.268,E2 23954.268} C_VEL
LIN {X 0,Y 503.563,Z 654.492,A -85,B 0,C 180,E1 23952.675,E2 23952.675} C_VEL
LIN {X 0,Y 501.928,Z 672.992,A -85,B 0,C 180,E1 23950.863,E2 23950.863} C_VEL
LIN {X 0,Y 500.52,Z 689.538,A -85,B 0,C 180,E1 23948.965,E2 23948.965} C_VEL
LIN {X 0,Y 499.191,Z 705.707,A -85,B 0,C 180,E1 23946.788,E2 23946.788} C_VEL
LIN {X 0,Y 498.148,Z 719.521,A -85,B 0,C 180,E1 23944.606,E2 23944.606} C_VEL
LIN {X 0,Y 497.299,Z 732.491,A -85,B 0,C 180,E1 23942.191,E2 23942.191} C_VEL
LIN {X 0,Y 496.7,Z 743.343,A -85,B 0,C 180,E1 23939.771,E2 23939.771} C_VEL
LIN {X 0,Y 496.307,Z 752.331,A -85,B 0,C 180,E1 23937.346,E2 23937.346} C_VEL
LIN {X 0,Y 496.078,Z 759.544,A -85,B 0,C 180,E1 23934.914,E2 23934.914} C_VEL
LIN {X 0,Y 495.969,Z 765.173,A -85,B 0,C 180,E1 23932.472,E2 23932.472} C_VEL
LIN {X 0,Y 495.912,Z 769.174,A -85,B 0,C 180,E1 23930.017,E2 23930.017} C_VEL
LIN {X 0,Y 495.908,Z 771.717,A -85,B 0,C 180,E1 23927.384,E2 23927.384} C_VEL
LIN {X 0,Y 495.913,Z 772.499,A -85,B 0,C 180,E1 23924.927,E2 23924.927} C_VEL
LIN {X 0,Y 495.908,Z 771.633,A -85,B 0,C 180,E1 23922.398,E2 23922.398} C_VEL
LIN {X 0,Y 495.915,Z 769.097,A -85,B 0,C 180,E1 23919.835,E2 23919.835} C_VEL
LIN {X 0,Y 495.959,Z 765.007,A -85,B 0,C 180,E1 23917.355,E2 23917.355} C_VEL
LIN {X 0,Y 496.097,Z 759.074,A -85,B 0,C 180,E1 23914.816,E2 23914.816} C_VEL
LIN {X 0,Y 496.334,Z 751.769,A -85,B 0,C 180,E1 23912.4,E2 23912.4} C_VEL
LIN {X 0,Y 496.739,Z 742.461,A -85,B 0,C 180,E1 23909.923,E2 23909.923} C_VEL
LIN {X 0,Y 497.347,Z 731.611,A -85,B 0,C 180,E1 23907.539,E2 23907.539} C_VEL
LIN {X 0,Y 498.234,Z 718.423,A -85,B 0,C 180,E1 23905.117,E2 23905.117} C_VEL
LIN {X 0,Y 499.294,Z 704.4,A -85,B 0,C 180,E1 23902.935,E2 23902.935} C_VEL
LIN {X 0,Y 500.624,Z 688.364,A -85,B 0,C 180,E1 23900.799,E2 23900.799} C_VEL
LIN {X 0,Y 502.118,Z 670.889,A -85,B 0,C 180,E1 23898.826,E2 23898.826} C_VEL
LIN {X 0,Y 503.696,Z 652.904,A -85,B 0,C 180,E1 23897.092,E2 23897.092} C_VEL
LIN {X 0,Y 505.405,Z 632.823,A -85,B 0,C 180,E1 23895.463,E2 23895.463} C_VEL
LIN {X 0,Y 506.959,Z 613.065,A -85,B 0,C 180,E1 23894.122,E2 23894.122} C_VEL
LIN {X 0,Y 508.055,Z 598.161,A -85,B 0,C 180,E1 23893.265,E2 23893.265} C_VEL
LIN {X 0,Y 507.704,Z 591.313,A -85,B 0,C 180,E1 23892.852,E2 23892.852} C_VEL
LIN {X 0,Y 503.638,Z 574.342,A -85,B 0,C 180,E1 23891.718,E2 23891.718} C_VEL
LIN {X 0,Y 503.202,Z 567.217,A -85,B 0,C 180,E1 23891.379,E2 23891.379} C_VEL
LIN {X 0,Y 504.256,Z 546.013,A -85,B 0,C 180,E1 23890.691,E2 23890.691} C_VEL
LIN {X 0,Y 505.052,Z 523.36,A -85,B 0,C 180,E1 23890.179,E2 23890.179} C_VEL
LIN {X 0,Y 507.879,Z 354.806,A -85,B 0,C 180,E1 23887.481,E2 23887.481} C_VEL
LIN {X 0,Y 508.998,Z 284.375,A -85,B 0,C 180,E1 23886.337,E2 23886.337} C_VEL
LIN {X 0,Y 497.058,Z 265.481,A -85,B 0,C 180,E1 23884.862,E2 23884.862} C_VEL
LIN {X 0,Y 491.877,Z 257.368,A -85,B 0,C 180,E1 23884.186,E2 23884.186} C_VEL
LIN {X 0,Y 489.396,Z 254.019,A -85,B 0,C 180,E1 23883.866,E2 23883.866} C_VEL
LIN {X 0,Y 488.815,Z 251.848,A -85,B 0,C 180,E1 23883.735,E2 23883.735} C_VEL
LIN {X 0,Y 488.794,Z 251.849,A -85,B 0,C 180,E1 23880.213,E2 23880.213} C_VEL
LIN {X 0,Y 488.81,Z 251.848,A -85,B 0,C 180,E1 23876.641,E2 23876.641} C_VEL
LIN {X 0,Y 488.836,Z 251.843,A -85,B 0,C 180,E1 23873.124,E2 23873.124} C_VEL
LIN {X 0,Y 488.806,Z 251.845,A -85,B 0,C 180,E1 23869.602,E2 23869.602} C_VEL
LIN {X 0,Y 488.788,Z 251.846,A -85,B 0,C 180,E1 23866.032,E2 23866.032} C_VEL
LIN {X 0,Y 488.809,Z 251.848,A -85,B 0,C 180,E1 23862.524,E2 23862.524} C_VEL
LIN {X 0,Y 488.834,Z 251.845,A -85,B 0,C 180,E1 23858.932,E2 23858.932} C_VEL
LIN {X 0,Y 488.801,Z 251.841,A -85,B 0,C 180,E1 23855.4,E2 23855.4} C_VEL
LIN {X 0,Y 488.782,Z 251.843,A -85,B 0,C 180,E1 23851.877,E2 23851.877} C_VEL
LIN {X 0,Y 488.816,Z 251.843,A -85,B 0,C 180,E1 23848.477,E2 23848.477} C_VEL
LIN {X 0,Y 488.822,Z 251.837,A -85,B 0,C 180,E1 23844.924,E2 23844.924} C_VEL
LIN {X 0,Y 488.782,Z 251.841,A -85,B 0,C 180,E1 23841.532,E2 23841.532} C_VEL
LIN {X 0,Y 488.784,Z 251.845,A -85,B 0,C 180,E1 23837.89,E2 23837.89} C_VEL
LIN {X 0,Y 488.828,Z 251.841,A -85,B 0,C 180,E1 23834.438,E2 23834.438} C_VEL
LIN {X 0,Y 488.805,Z 251.844,A -85,B 0,C 180,E1 23830.898,E2 23830.898} C_VEL
LIN {X 0,Y 488.774,Z 251.847,A -85,B 0,C 180,E1 23827.511,E2 23827.511} C_VEL
LIN {X 0,Y 488.802,Z 251.849,A -85,B 0,C 180,E1 23824.042,E2 23824.042} C_VEL
LIN {X 0,Y 488.816,Z 251.843,A -85,B 0,C 180,E1 23820.601,E2 23820.601} C_VEL
LIN {X 0,Y 488.772,Z 251.843,A -85,B 0,C 180,E1 23817.175,E2 23817.175} C_VEL
LIN {X 0,Y 488.777,Z 251.845,A -85,B 0,C 180,E1 23813.615,E2 23813.615} C_VEL
LIN {X 0,Y 488.829,Z 251.85,A -85,B 0,C 180,E1 23810.194,E2 23810.194} C_VEL
LIN {X 0,Y 488.782,Z 251.848,A -85,B 0,C 180,E1 23806.735,E2 23806.735} C_VEL
LIN {X 0,Y 488.766,Z 251.848,A -85,B 0,C 180,E1 23803.256,E2 23803.256} C_VEL
LIN {X 0,Y 488.802,Z 251.845,A -85,B 0,C 180,E1 23799.807,E2 23799.807} C_VEL
LIN {X 0,Y 488.794,Z 251.849,A -85,B 0,C 180,E1 23796.382,E2 23796.382} C_VEL
LIN {X 0,Y 488.76,Z 251.85,A -85,B 0,C 180,E1 23792.964,E2 23792.964} C_VEL
LIN {X 0,Y 488.787,Z 251.849,A -85,B 0,C 180,E1 23789.534,E2 23789.534} C_VEL
LIN {X 0,Y 488.791,Z 251.847,A -85,B 0,C 180,E1 23786.219,E2 23786.219} C_VEL
LIN {X 0,Y 488.756,Z 251.849,A -85,B 0,C 180,E1 23782.743,E2 23782.743} C_VEL
LIN {X 0,Y 488.77,Z 251.849,A -85,B 0,C 180,E1 23779.227,E2 23779.227} C_VEL
LIN {X 0,Y 488.816,Z 251.849,A -85,B 0,C 180,E1 23775.784,E2 23775.784} C_VEL
LIN {X 0,Y 488.755,Z 251.85,A -85,B 0,C 180,E1 23772.402,E2 23772.402} C_VEL
LIN {X 0,Y 488.752,Z 251.851,A -85,B 0,C 180,E1 23768.824,E2 23768.824} C_VEL
LIN {X 0,Y 488.807,Z 251.851,A -85,B 0,C 180,E1 23765.515,E2 23765.515} C_VEL
LIN {X 0,Y 488.771,Z 251.851,A -85,B 0,C 180,E1 23761.991,E2 23761.991} C_VEL
LIN {X 0,Y 488.75,Z 251.851,A -85,B 0,C 180,E1 23758.592,E2 23758.592} C_VEL
LIN {X 0,Y 488.793,Z 251.847,A -85,B 0,C 180,E1 23755.188,E2 23755.188} C_VEL
LIN {X 0,Y 488.772,Z 251.85,A -85,B 0,C 180,E1 23751.884,E2 23751.884} C_VEL
LIN {X 0,Y 488.755,Z 251.848,A -85,B 0,C 180,E1 23748.434,E2 23748.434} C_VEL
LIN {X 0,Y 488.8,Z 251.848,A -85,B 0,C 180,E1 23745.063,E2 23745.063} C_VEL
LIN {X 0,Y 488.784,Z 251.85,A -85,B 0,C 180,E1 23741.637,E2 23741.637} C_VEL
LIN {X 0,Y 488.758,Z 251.848,A -85,B 0,C 180,E1 23738.236,E2 23738.236} C_VEL
LIN {X 0,Y 488.794,Z 251.845,A -85,B 0,C 180,E1 23734.818,E2 23734.818} C_VEL
LIN {X 0,Y 488.806,Z 251.849,A -85,B 0,C 180,E1 23731.341,E2 23731.341} C_VEL
LIN {X 0,Y 488.764,Z 251.85,A -85,B 0,C 180,E1 23728.005,E2 23728.005} C_VEL
LIN {X 0,Y 488.782,Z 251.85,A -85,B 0,C 180,E1 23724.481,E2 23724.481} C_VEL
LIN {X 0,Y 488.835,Z 251.844,A -85,B 0,C 180,E1 23720.95,E2 23720.95} C_VEL
LIN {X 0,Y 488.778,Z 251.854,A -85,B 0,C 180,E1 23717.541,E2 23717.541} C_VEL
LIN {X 0,Y 488.79,Z 252.004,A -85,B 0,C 180,E1 23715.932,E2 23715.932} C_VEL
LIN {X 0,Y 490.244,Z 255.561,A -85,B 0,C 180,E1 23715.444,E2 23715.444} C_VEL
LIN {X 0,Y 497.932,Z 272.526,A -85,B 0,C 180,E1 23713.12,E2 23713.12} C_VEL
LIN {X 0,Y 505.744,Z 290.691,A -85,B 0,C 180,E1 23710.83,E2 23710.83} C_VEL
LIN {X 0,Y 505.318,Z 300.969,A -85,B 0,C 180,E1 23710.056,E2 23710.056} C_VEL
LIN {X 0,Y 509.518,Z 326.675,A -85,B 0,C 180,E1 23709.172,E2 23709.172} C_VEL
LIN {X 0,Y 506.212,Z 522.23,A -85,B 0,C 180,E1 23706.036,E2 23706.036} C_VEL
LIN {X 0,Y 504.845,Z 607.372,A -85,B 0,C 180,E1 23704.681,E2 23704.681} C_VEL
LIN {X 0,Y 503.982,Z 629.092,A -85,B 0,C 180,E1 23704.15,E2 23704.15} C_VEL
LIN {X 0,Y 502.879,Z 650.83,A -85,B 0,C 180,E1 23703.417,E2 23703.417} C_VEL
LIN {X 0,Y 501.613,Z 671.863,A -85,B 0,C 180,E1 23702.497,E2 23702.497} C_VEL
LIN {X 0,Y 500.158,Z 690.758,A -85,B 0,C 180,E1 23701.449,E2 23701.449} C_VEL
LIN {X 0,Y 498.539,Z 709.997,A -85,B 0,C 180,E1 23700.164,E2 23700.164} C_VEL
LIN {X 0,Y 496.909,Z 727.867,A -85,B 0,C 180,E1 23698.743,E2 23698.743} C_VEL
LIN {X 0,Y 495.213,Z 745.73,A -85,B 0,C 180,E1 23697.076,E2 23697.076} C_VEL
LIN {X 0,Y 493.634,Z 762.53,A -85,B 0,C 180,E1 23695.25,E2 23695.25} C_VEL
LIN {X 0,Y 492.245,Z 777.659,A -85,B 0,C 180,E1 23693.332,E2 23693.332} C_VEL
LIN {X 0,Y 491.006,Z 791.791,A -85,B 0,C 180,E1 23691.25,E2 23691.25} C_VEL
LIN {X 0,Y 489.953,Z 805.285,A -85,B 0,C 180,E1 23688.932,E2 23688.932} C_VEL
LIN {X 0,Y 489.176,Z 816.687,A -85,B 0,C 180,E1 23686.626,E2 23686.626} C_VEL
LIN {X 0,Y 488.607,Z 826.6,A -85,B 0,C 180,E1 23684.214,E2 23684.214} C_VEL
LIN {X 0,Y 488.245,Z 835.12,A -85,B 0,C 180,E1 23681.696,E2 23681.696} C_VEL
LIN {X 0,Y 488.049,Z 841.875,A -85,B 0,C 180,E1 23679.194,E2 23679.194} C_VEL
LIN {X 0,Y 487.948,Z 846.815,A -85,B 0,C 180,E1 23676.706,E2 23676.706} C_VEL
LIN {X 0,Y 487.914,Z 850.334,A -85,B 0,C 180,E1 23674.112,E2 23674.112} C_VEL
LIN {X 0,Y 487.9,Z 852.085,A -85,B 0,C 180,E1 23671.76,E2 23671.76} C_VEL
LIN {X 0,Y 487.901,Z 852.372,A -85,B 0,C 180,E1 23669.294,E2 23669.294} C_VEL
LIN {X 0,Y 487.915,Z 851.233,A -85,B 0,C 180,E1 23666.827,E2 23666.827} C_VEL
LIN {X 0,Y 487.931,Z 848.457,A -85,B 0,C 180,E1 23664.354,E2 23664.354} C_VEL
LIN {X 0,Y 488.004,Z 843.861,A -85,B 0,C 180,E1 23661.733,E2 23661.733} C_VEL
LIN {X 0,Y 488.152,Z 837.933,A -85,B 0,C 180,E1 23659.257,E2 23659.257} C_VEL
LIN {X 0,Y 488.425,Z 830.474,A -85,B 0,C 180,E1 23656.865,E2 23656.865} C_VEL
LIN {X 0,Y 488.917,Z 820.835,A -85,B 0,C 180,E1 23654.338,E2 23654.338} C_VEL
LIN {X 0,Y 489.594,Z 810.347,A -85,B 0,C 180,E1 23652.038,E2 23652.038} C_VEL
LIN {X 0,Y 490.527,Z 797.754,A -85,B 0,C 180,E1 23649.725,E2 23649.725} C_VEL
LIN {X 0,Y 491.697,Z 783.705,A -85,B 0,C 180,E1 23647.523,E2 23647.523} C_VEL
LIN {X 0,Y 493.106,Z 768.194,A -85,B 0,C 180,E1 23645.437,E2 23645.437} C_VEL
LIN {X 0,Y 494.629,Z 752.05,A -85,B 0,C 180,E1 23643.573,E2 23643.573} C_VEL
LIN {X 0,Y 496.253,Z 734.751,A -85,B 0,C 180,E1 23641.87,E2 23641.87} C_VEL
LIN {X 0,Y 498.02,Z 715.73,A -85,B 0,C 180,E1 23640.27,E2 23640.27} C_VEL
LIN {X 0,Y 499.693,Z 696.696,A -85,B 0,C 180,E1 23638.916,E2 23638.916} C_VEL
LIN {X 0,Y 501.165,Z 677.845,A -85,B 0,C 180,E1 23637.812,E2 23637.812} C_VEL
LIN {X 0,Y 502.396,Z 658.77,A -85,B 0,C 180,E1 23636.916,E2 23636.916} C_VEL
LIN {X 0,Y 503.457,Z 636.932,A -85,B 0,C 180,E1 23636.12,E2 23636.12} C_VEL
LIN {X 0,Y 504.339,Z 614.82,A -85,B 0,C 180,E1 23635.53,E2 23635.53} C_VEL
LIN {X 0,Y 504.929,Z 588.867,A -85,B 0,C 180,E1 23635.066,E2 23635.066} C_VEL
LIN {X 0,Y 507.15,Z 424.72,A -85,B 0,C 180,E1 23632.521,E2 23632.521} C_VEL
LIN {X 0,Y 508.825,Z 324.498,A -85,B 0,C 180,E1 23630.858,E2 23630.858} C_VEL
LIN {X 0,Y 504.002,Z 294.328,A -85,B 0,C 180,E1 23629.799,E2 23629.799} C_VEL
LIN {X 0,Y 504.011,Z 288.759,A -85,B 0,C 180,E1 23629.36,E2 23629.36} C_VEL
LIN {X 0,Y 493.814,Z 263.414,A -85,B 0,C 180,E1 23626.29,E2 23626.29} C_VEL
LIN {X 0,Y 489.984,Z 255.111,A -85,B 0,C 180,E1 23625.08,E2 23625.08} C_VEL
LIN {X 0,Y 488.781,Z 251.853,A -85,B 0,C 180,E1 23624.56,E2 23624.56} C_VEL
